# B&R Automation Studio project Panasonic_LinkaKapacitorov_A2021040 (part 3)

#### OvlRucnejCitackyQR.st
```iecst
ACTION OvlRucnejCitackyQR:

	//"$L"  LF - linefeed - skok na druhý riadok

	CASE RucCitackaQR.Step OF

		0://Nulovanie//
			RucCitackaQR.Command.PrimajData:= FALSE;
			RucCitackaQR.Command.ZatvorKomunikaciu:= FALSE;
			RucCitackaQR.Command.PotvrdeniePoruchy:= FALSE;
			RucCitackaQR.Status.PoruchaOtvoreniaKomunikacie:= FALSE;
			RucCitackaQR.Status.PoruchaZatvoreniaKomunikacie:= FALSE;
			RucCitackaQR.Status.PoruchaCitaniaDat:= FALSE;
			RucCitackaQR.Status.PoruchaUvolneniaRECEIVE_Buffera:= FALSE;
			RucCitackaQR.Step:= 1;

		1://Rozhodnutie o činnosti//
			IF RucCitackaQR.Command.PrimajData THEN
				RucCitackaQR.Step:= 10;
			ELSIF Linka.CitackaQRkodu_AKTIVNA THEN
				RucCitackaQR.Step:= 10;
			END_IF

		10://Prímanie dát - otvorenie seriovej komunikácie//
			RucCitackaQR.FRM_xopen_0.enable:= TRUE;
			RucCitackaQR.FRM_xopen_0.device:=  ADR('IF1');
			RucCitackaQR.FRM_xopen_0.mode:= ADR('/PHY=RS232 /BD=115200 /DB=8 /PA=N /SB=1');
			RucCitackaQR.FRM_xopen_0.config:= ADR(RucCitackaQR.xopenConfig);

			RucCitackaQR.xopenConfig.idle:= 100;
			RucCitackaQR.xopenConfig.delimc:= 0;
			RucCitackaQR.xopenConfig.delim[0]:= 0;
			RucCitackaQR.xopenConfig.delim[1]:= 0;
			RucCitackaQR.xopenConfig.tx_cnt:= 3;
			RucCitackaQR.xopenConfig.rx_cnt:= 3;
			RucCitackaQR.xopenConfig.tx_len:= 256;
			RucCitackaQR.xopenConfig.rx_len:= 256;
			RucCitackaQR.xopenConfig.argc:= 0;
			RucCitackaQR.xopenConfig.argv:= 0;

			RucCitackaQR.FRM_xopen_0();

			IF RucCitackaQR.FRM_xopen_0.status = 0 THEN   //Otvorenie komunikácie prebehlo OK
				RucCitackaQR.Step:= 11;
			ELSIF RucCitackaQR.FRM_xopen_0.status = 65535 THEN  //Prebieha otvorenie komunikácie - stav BUSY
				RucCitackaQR.Step:= 10;
			ELSE
				RucCitackaQR.Status.PoruchaOtvoreniaKomunikacie:= TRUE;
				RucCitackaQR.Step:= 100;  //Porucha otvorenia komunikácie
			END_IF

		11://Prímanie dát - čítanie dát z komunikácie//
			RucCitackaQR.FRM_read_0.enable:= TRUE;
			RucCitackaQR.FRM_read_0.ident:= RucCitackaQR.FRM_xopen_0.ident;
			RucCitackaQR.FRM_read_0();

			IF RucCitackaQR.FRM_read_0.status = 0 THEN //Čítanie dát z komunikácie prebehlo OK
				RucCitackaQR.Step:= 12;
			ELSIF RucCitackaQR.Command.ZatvorKomunikaciu THEN
				RucCitackaQR.Step:= 0;
			ELSIF NOT Linka.CitackaQRkodu_AKTIVNA THEN
				RucCitackaQR.Step:= 0;
			ELSIF RucCitackaQR.FRM_read_0.status = 60 THEN //Prebieha čítanie dát z komunikácie - stav žiadne dáta
				RucCitackaQR.Step:= 11;
			ELSIF RucCitackaQR.FRM_read_0.status = 8079 THEN //Prišli zlé alebo neúplné dáta
				RucCitackaQR.Step:= 18;
			ELSE
				RucCitackaQR.Status.PoruchaCitaniaDat:= TRUE;
				RucCitackaQR.Step:= 100;  //Porucha čítania dát z komunikácie
			END_IF

		12://Prímanie dát - kopírovanie dát do RECEIVE buffera//
			brsmemset(ADR(RucCitackaQR.PrecitaneData),0,SIZEOF(RucCitackaQR.PrecitaneData)); //Vynulovanie prečítanej správy
			brsmemcpy(ADR(RucCitackaQR.PrecitaneData),RucCitackaQR.FRM_read_0.buffer,RucCitackaQR.FRM_read_0.buflng); //Zkopírovanie dát z RECEIVE buffera do prečítanej správy
			RucCitackaQR.Step:= 18;

		18://Prímanie dát - uvolnenie RECEIVE buffera//
			RucCitackaQR.FRM_rbuf_0.enable:= TRUE;
			RucCitackaQR.FRM_rbuf_0.buffer:= RucCitackaQR.FRM_read_0.buffer;
			RucCitackaQR.FRM_rbuf_0.buflng:= RucCitackaQR.FRM_read_0.buflng;
			RucCitackaQR.FRM_rbuf_0.ident:= RucCitackaQR.FRM_xopen_0.ident;
			RucCitackaQR.FRM_rbuf_0();

			IF RucCitackaQR.FRM_rbuf_0.status = 0 THEN //Uvolnenie RECEIVE buffera prebehlo OK
				IF RucCitackaQR.Command.ZatvorKomunikaciu THEN
					RucCitackaQR.Step:= 20;
				ELSE
					RucCitackaQR.Step:= 11;
				END_IF
			ELSIF RucCitackaQR.FRM_rbuf_0.status = 65535 THEN //Prebieha uvolnenie RECEIVE buffera - stav BUSY
				RucCitackaQR.Step:= 18;
			ELSIF RucCitackaQR.FRM_rbuf_0.status = 8072 THEN //Buffer je poškodený - op)tovné čítanie
				RucCitackaQR.Step:= 11;
			ELSE
				RucCitackaQR.Status.PoruchaUvolneniaRECEIVE_Buffera:= TRUE;
				RucCitackaQR.Step:= 100;  //Porucha uvolnenia RECEIVE buffera
			END_IF

		20://Prímanie dát - zatvorenie komunikácie//
			RucCitackaQR.FRM_close_0.enable:= TRUE;
			RucCitackaQR.FRM_close_0.ident:= RucCitackaQR.FRM_xopen_0.ident;
			RucCitackaQR.FRM_close_0();

			IF RucCitackaQR.FRM_close_0.status = 0 THEN //Zatvorenie komunikácie prebehlo OK
				RucCitackaQR.Step:= 0;
			ELSIF RucCitackaQR.FRM_close_0.status = 65535 THEN //Prebieha zatvorenie komunikácie - stav BUSY
				RucCitackaQR.Step:= 20;
			ELSE
				RucCitackaQR.Status.PoruchaZatvoreniaKomunikacie:= TRUE;
				RucCitackaQR.Step:= 100;  //Porucha zatvorenia komunikácie
			END_IF

		100://Porucha komunikácie//
			IF RucCitackaQR.Command.PotvrdeniePoruchy THEN
				RucCitackaQR.Step:= 0;
			END_IF

	END_CASE

END_ACTION
```

#### ZmenaModelu.st
```iecst
ACTION ZmenaModelu:

		//***********************************************Zobrazenie stavov zmeny modelu***********************************************//
    //0 - Čakám na zmenu modelu.
    //1 - Nebol načítaný názov modelu !!!
    //2 - Nebol načítaný LOT !!!
    //3 - Zmena modelu prebehla OK !!!
	//4 - Zadaný model nieje v databázi linky !!!

	//Farba pozadia//
	//0 - sivá
	//1 - modrá
	//2 - zelená
	//3 - červená

	IF EDGEPOS(Vizu.CisloAktualnejObrazovky = 4)THEN
		Vizu.StavZmenyModelu_Index:= 0;
		Vizu.StavZmenyModelu_Farba:= 0;
		Vizu.Nacitany_MODEL:= '';
		Vizu.Nacitany_LOT:= '';
	END_IF

	//Zistenie počtu načítaných znakov//
	PocetNacitanychZnakov := brsstrlen(ADR(RucCitackaQR.PrecitaneData)); //Zistenie počtu znakov vstupnej spravy

	//Zistenie či sa jedná o Názov modelu alebo číslo Lotu//
	brsmemcpy(ADR(NacitaneZnaky_POLE),ADR(RucCitackaQR.PrecitaneData),SIZEOF(RucCitackaQR.PrecitaneData)); //Vyplnenie polia znakmy vstupnej správy

	//Zapísanie načítanej hodnoty do pola Nazov Modelu alebo Cislo Lotu// EZT
	IF RucCitackaQR.PrecitaneData <> '' THEN
		IF NacitaneZnaky_POLE[0] = 69 AND NacitaneZnaky_POLE[1] = 90 AND NacitaneZnaky_POLE[2] = 84 AND PocetNacitanychZnakov = 12 THEN
			Vizu.Nacitany_MODEL:= RucCitackaQR.PrecitaneData;
		ELSIF NacitaneZnaky_POLE[0] = 66 AND PocetNacitanychZnakov = 11 THEN
			Vizu.Nacitany_LOT:= RucCitackaQR.PrecitaneData;
		END_IF
		RucCitackaQR.PrecitaneData:= '';
	END_IF

	CASE SC_ZmenaModelu.Step OF

		0://Vynulovanie uživatela//
			SC_ZmenaModelu.StepName:= '0 - Nulovanie';
			Linka.ZmenModel:= FALSE;
			i:= 0;
			SC_ZmenaModelu.ResetStep:= TRUE;
			SC_ZmenaModelu.Step:= 1;

		1://Rozhodnutie o činnosti//
			SC_ZmenaModelu.StepName:= '1 - Rozhodnutie o cinnosti';
			IF Linka.ZmenModel THEN
				SC_ZmenaModelu.Step:= 10;
			END_IF

		10://Kontrola zadania modelu//
			SC_ZmenaModelu.StepName:= '10 - Kontrola zadania modelu';
			IF Vizu.Nacitany_MODEL <> '' AND Vizu.Nacitany_LOT <> '' THEN
				SC_ZmenaModelu.ResetStep:= TRUE;
				SC_ZmenaModelu.Step:= 11;
			ELSE
				IF Vizu.Nacitany_MODEL = '' THEN
					Vizu.StavZmenyModelu_Index:= 1;
					Vizu.StavZmenyModelu_Farba:= 3;
				ELSIF Vizu.Nacitany_LOT = '' THEN
					Vizu.StavZmenyModelu_Index:= 2;
					Vizu.StavZmenyModelu_Farba:= 3;
				END_IF
				SC_ZmenaModelu.ResetStep:= TRUE;
				SC_ZmenaModelu.Step:= 0;
			END_IF

		11://Hladanie modelu v recepturach//
			SC_ZmenaModelu.StepName:= '11 - Hladanie modelu v recepturach';
			ModelNajdeny:= FALSE;
			FOR i:= 0 TO 150 BY 1 DO
				IF (Receptura[i].NazovModelu = Vizu.Nacitany_MODEL) AND NOT ModelNajdeny THEN
					HistoriaVyroby[IndexHistorie].NazovModelu:= Zvoleny_MODEL;
					HistoriaVyroby[IndexHistorie].NazovLOTU:= Zvoleny_LOT;
					HistoriaVyroby[IndexHistorie].PocetVyrobenychKusov_OK:= PocetVyrobenychKusov_OK;
					HistoriaVyroby[IndexHistorie].PocetVyrobenychKusov_NG:= PocetVyrobenychKusov_NG;
					HistoriaVyroby[IndexHistorie].Pomer_OK_kusov_IDR:= Pomer_OK_kusov_IDR;
					IndexHistorie:= IndexHistorie + 1;
					IF IndexHistorie > 5 THEN
						IndexHistorie:= 0;
					END_IF
					Linka.PAR.Zvoleny_MODEL:= Vizu.Nacitany_MODEL;
					Zvoleny_MODEL:= Vizu.Nacitany_MODEL;
					Linka.PAR.Zvoleny_LOT:= Vizu.Nacitany_LOT;
					Zvoleny_LOT:= Vizu.Nacitany_LOT;
					Linka.PAR.IndexZvoleneReceptury:= i;
					Vizu.StavZmenyModelu_Index:= 3;
					Vizu.StavZmenyModelu_Farba:= 2;
					RESET_PoctuVyrobenychKusov:= TRUE;
					Linka.Rezim_BezCistenia:= FALSE;
					Linka.Rezim_BezTlaceEtikety:= FALSE;
					Linka.Rezim_Testovania:= FALSE;
					NacitajRecepturu:= TRUE;
					ModelNajdeny:= TRUE;
				END_IF
			END_FOR
			IF NOT ModelNajdeny THEN
				Vizu.StavZmenyModelu_Index:= 4;
				Vizu.StavZmenyModelu_Farba:= 3;
			END_IF
			SC_ZmenaModelu.ResetStep:= TRUE;
			SC_ZmenaModelu.Step:= 0;

	END_CASE

END_ACTION
```

### Program Logical/Program/KontrolaOtacaniaTrysiek (IEC)

#### Main.st - Init, cyclic, exit code
```iecst
PROGRAM _INIT
	(* Insert code here *)

END_PROGRAM

PROGRAM _CYCLIC

	//Volanie funkcie SequenceControl//
	SequenceControl(SC:= SC_OvlCistenia);

	CASE SC_OvlCistenia.Step OF

		0:
			SC_OvlCistenia.StepName:='0 - Nulovanie';
			CasOtacaniaHornejTrisky_1.IN:= FALSE;
			CasOtacaniaHornejTrisky_2.IN:= FALSE;
			CasOtacaniaHornejTrisky_3.IN:= FALSE;
			CasOtacaniaHornejTrisky_4.IN:= FALSE;
			CasOtacaniaSpodnejTrisky_1.IN:= FALSE;
			CasOtacaniaSpodnejTrisky_2.IN:= FALSE;
			CasOtacaniaSpodnejTrisky_3.IN:= FALSE;
			Linka.OUT.IonJednotka_START:= FALSE;
			Linka.OUT.IonJednotka_AIR:= FALSE;
			SC_OvlCistenia.ResetStep:= TRUE;
			SC_OvlCistenia.Step:= 1;

		1:
			SC_OvlCistenia.StepName:='1 - Cakam na spustenie cistenia';

			IF Linka.OUT.IonJednotka_START THEN
				SC_OvlCistenia.Step:= 10;
			END_IF

		10:
			SC_OvlCistenia.StepName:='10 - spustenie kontroly otacania trisiek';
			SC_OvlCistenia.IdleTime.PT:= T#2s;
			SC_OvlCistenia.AlarmTime.PT:= T#1s;

			Linka.OUT.IonJednotka_AIR:= TRUE;

			SC_OvlCistenia.IdleTime.IN:= TRUE;

			IF EDGE(Linka.IN.SnimacRotacieHornTrysiek_1_IS7) THEN
				CasOtacaniaHornejTrisky_1.IN:= FALSE;
			ELSE
				CasOtacaniaHornejTrisky_1.IN:= TRUE;
			END_IF

			IF EDGE(Linka.IN.SnimacRotacieHornTrysiek_2_IS8) THEN
				CasOtacaniaHornejTrisky_2.IN:= FALSE;
			ELSE
				CasOtacaniaHornejTrisky_2.IN:= TRUE;
			END_IF

			IF EDGE(Linka.IN.SnimacRotacieHornTrysiek_3_IS9) THEN
				CasOtacaniaHornejTrisky_3.IN:= FALSE;
			ELSE
				CasOtacaniaHornejTrisky_3.IN:= TRUE;
			END_IF

			IF EDGE(Linka.IN.SnimacRotacieHornTrysiek_4_IS10) THEN
				CasOtacaniaHornejTrisky_4.IN:= FALSE;
			ELSE
				CasOtacaniaHornejTrisky_4.IN:= TRUE;
			END_IF

			IF EDGE(Linka.IN.SnimacRotacieSpodTrysiek_1_IS11) THEN
				CasOtacaniaSpodnejTrisky_1.IN:= FALSE;
			ELSE
				CasOtacaniaSpodnejTrisky_1.IN:= TRUE;
			END_IF

			IF EDGE(Linka.IN.SnimacRotacieSpodTrysiek_2_IS12) THEN
				CasOtacaniaSpodnejTrisky_2.IN:= FALSE;
			ELSE
				CasOtacaniaSpodnejTrisky_2.IN:= TRUE;
			END_IF

			IF EDGE(Linka.IN.SnimacRotacieSpodTrysiek_3_IS13) THEN
				CasOtacaniaSpodnejTrisky_3.IN:= FALSE;
			ELSE
				CasOtacaniaSpodnejTrisky_3.IN:= TRUE;
			END_IF

			IF NOT Linka.OUT.IonJednotka_START THEN
				SC_OvlCistenia.ResetStep:= TRUE;
				SC_OvlCistenia.Step:= 0;
			END_IF

			IF SC_OvlCistenia.IdleTime.Q THEN
				IF CasOtacaniaHornejTrisky_1.Q THEN
					Alarmy[37]:= TRUE;
					Linka.STAV.PoruchaOtacaniaTrysiek:= TRUE;
					SC_OvlCistenia.ResetStep:= TRUE;
					SC_OvlCistenia.Step:= 0;
				ELSIF CasOtacaniaHornejTrisky_2.Q THEN
					Alarmy[37]:= TRUE;
					Linka.STAV.PoruchaOtacaniaTrysiek:= TRUE;
					SC_OvlCistenia.ResetStep:= TRUE;
					SC_OvlCistenia.Step:= 0;
				ELSIF CasOtacaniaHornejTrisky_3.Q THEN
					Alarmy[37]:= TRUE;
					Linka.STAV.PoruchaOtacaniaTrysiek:= TRUE;
					SC_OvlCistenia.ResetStep:= TRUE;
					SC_OvlCistenia.Step:= 0;
				ELSIF CasOtacaniaHornejTrisky_4.Q THEN
					Alarmy[37]:= TRUE;
					Linka.STAV.PoruchaOtacaniaTrysiek:= TRUE;
					SC_OvlCistenia.ResetStep:= TRUE;
					SC_OvlCistenia.Step:= 0;
				ELSIF CasOtacaniaSpodnejTrisky_1.Q THEN
					Alarmy[38]:= TRUE;
					Linka.STAV.PoruchaOtacaniaTrysiek:= TRUE;
					SC_OvlCistenia.ResetStep:= TRUE;
					SC_OvlCistenia.Step:= 0;
				ELSIF CasOtacaniaSpodnejTrisky_2.Q THEN
					Alarmy[38]:= TRUE;
					Linka.STAV.PoruchaOtacaniaTrysiek:= TRUE;
					SC_OvlCistenia.ResetStep:= TRUE;
					SC_OvlCistenia.Step:= 0;
				ELSIF CasOtacaniaSpodnejTrisky_3.Q THEN
					Alarmy[38]:= TRUE;
					Linka.STAV.PoruchaOtacaniaTrysiek:= TRUE;
					SC_OvlCistenia.ResetStep:= TRUE;
					SC_OvlCistenia.Step:= 0;
				END_IF
			END_IF

	END_CASE

	CasOtacaniaHornejTrisky_1.PT:= T#300ms;
	CasOtacaniaHornejTrisky_1();
	CasOtacaniaHornejTrisky_2.PT:= T#300ms;
	CasOtacaniaHornejTrisky_2();
	CasOtacaniaHornejTrisky_3.PT:= T#300ms;
	CasOtacaniaHornejTrisky_3();
	CasOtacaniaHornejTrisky_4.PT:= T#300ms;
	CasOtacaniaHornejTrisky_4();
	CasOtacaniaSpodnejTrisky_1.PT:= T#500ms;
	CasOtacaniaSpodnejTrisky_1();
	CasOtacaniaSpodnejTrisky_2.PT:= T#500ms;
	CasOtacaniaSpodnejTrisky_2();
	CasOtacaniaSpodnejTrisky_3.PT:= T#500ms;
	CasOtacaniaSpodnejTrisky_3();

END_PROGRAM

PROGRAM _EXIT
	(* Insert code here *)

END_PROGRAM
```

#### Variables.var - Local variables
```iecst
VAR
	SC_OvlCistenia : SequenceControlTyp := (0);
	CasOtacaniaHornejTrisky_1 : TON := (0);
	CasOtacaniaHornejTrisky_2 : TON := (0);
	CasOtacaniaHornejTrisky_3 : TON := (0);
	CasOtacaniaHornejTrisky_4 : TON := (0);
	CasOtacaniaSpodnejTrisky_1 : TON := (0);
	CasOtacaniaSpodnejTrisky_2 : TON := (0);
	CasOtacaniaSpodnejTrisky_3 : TON := (0);
END_VAR
```

### Program Logical/Program/VstupnyVytah (IEC)

#### Main.st - Init, cyclic, exit code
```iecst
PROGRAM _INIT
	VstupVytah.PAR.Zdvih_ZadanaJoggRychlost:= 10;

END_PROGRAM

PROGRAM _CYCLIC

	//Volanie podprogramov//
	OvlMenica;
	OvlDveri;
	OvlCitackyRFID;

	//Volanie funkcie SequenceControl//
	SequenceControl(SC:= SC_VstupVytah);

	//Reset sekcie //
	IF VstupVytah.Reset THEN
		SC_VstupVytah.Step:= 0;
		VstupVytah.Reset:= FALSE;
	ELSIF NOT Safety.STAV.ZonaCS_AKTIVNA THEN
		SC_VstupVytah.Step:= 0;
	END_IF

	CASE SC_VstupVytah.Step OF

		0:
			SC_VstupVytah.StepName:='0 - Nulovanie';
			VstupVytah.Automat:= FALSE;
			VstupVytah.KoniecCyklu:= FALSE;
			VstupVytah.Manual:= FALSE;
			VstupVytah.STAV.PoINIT:= FALSE;
			SC_OvlMenica.Step:= 0;
			SC_OvlDveri.Step:= 0;
			VstupVytah.OUT.Dopravnik_ChodVPRED_ELR1:= FALSE;
			VstupVytah.OUT.Dopravnik_ChodVZAD_ELR1:= FALSE;
			VstupVytah.RR_Dopravnik_VPRED:= FALSE;
			VstupVytah.RR_Dopravnik_VZAD:= FALSE;
			IF PoruchaVstupnehoVytahu THEN
				VstupVytah.OUT.Banner_CervenaLED_IOS1:= Blikac200ms;
			ELSE
				VstupVytah.OUT.Banner_CervenaLED_IOS1:= FALSE;
			END_IF
			VstupVytah.OUT.Banner_ZelenaLED_IOS1:= FALSE;
			VstupVytah.STAV.PrebiehaVyvazaniePaletky:= FALSE;
			VstupVytah.STAV.VytahNapolohovany:= FALSE;
			Vizu.ZobrazHlasenie_NespravTypPaletky:= 1;
			VstupVytah.STAV.ObsluhaPotvrdilaBanner:= FALSE;
			VstupnyVytah_Statistika.IN.START_MeraniaCasu:= FALSE;

			IF Safety.STAV.ZonaCS_AKTIVNA AND Safety.STAV.ZonaVstupnyVytah_AKTIVNA AND Linka.IN.TlakVzduchu_OK_S2 AND NOT NastalaPorucha AND Linka.STAV.Hardware_OK THEN
				VstupVytah.OUT.Banner_CervenaLED_IOS1:= FALSE;
				SC_VstupVytah.ResetStep:= TRUE;
				SC_VstupVytah.Step:= 1;
			END_IF

		1:
			SC_VstupVytah.StepName:='1 - Cakam na spustenie vyroby';
			VstupVytah.KoniecCyklu:= FALSE;
			IF VstupVytah.Automat THEN
				SC_VstupVytah.Step:= 2;
			ELSIF VstupVytah.Manual THEN
				SC_VstupVytah.Step:= 700;
			END_IF

			//********************************************************Inicializácia****************************************************************************//

		2:
			SC_VstupVytah.StepName:='2 - Inicializacia - cakam na spustenie inicializacie';
			SC_VstupVytah.IdleTime.PT:= T#500ms;
			SC_VstupVytah.AlarmTime.PT:= T#5s;

			SC_VstupVytah.IdleTime.IN:= TRUE;

			IF SC_VstupVytah.IdleTime.Q THEN
				SC_VstupVytah.ResetStep:= TRUE;
				SC_VstupVytah.Step:= 5;
			END_IF

		5:
			SC_VstupVytah.StepName:='5 - Inicializacia - spustam dopravnik vytahu pre navezenie paletky';
			SC_VstupVytah.IdleTime.PT:= T#500ms;
			SC_VstupVytah.AlarmTime.PT:= T#7s;

			SC_VstupVytah.IdleTime.IN:= VstupVytah.IN.PritomnostPaletky_IS3;

			IF NOT SC_VstupVytah.Switch1 THEN
				VstupVytah.OUT.Dopravnik_ChodVZAD_ELR1:= TRUE;
				SC_VstupVytah.AlarmTime.IN:= TRUE;
				SC_VstupVytah.Switch1:= TRUE;
			END_IF

			IF SC_VstupVytah.IdleTime.Q AND NOT VstupVytah.IN.PrechodDopravnikaVytahu_OS1 THEN
				VstupVytah.OUT.Dopravnik_ChodVZAD_ELR1:= FALSE;
				SC_VstupVytah.ResetStep:= TRUE;
				SC_VstupVytah.Step:= 10;
			ELSIF SC_VstupVytah.AlarmTime.Q AND NOT VstupVytah.IN.PritomnostPaletky_IS3 AND NOT VstupVytah.IN.PrechodDopravnikaVytahu_OS1 THEN
				VstupVytah.OUT.Dopravnik_ChodVZAD_ELR1:= FALSE;
				SC_VstupVytah.ResetStep:= TRUE;
				SC_VstupVytah.Step:= 10;
			ELSIF SC_VstupVytah.AlarmTime.Q AND VstupVytah.IN.PrechodDopravnikaVytahu_OS1 THEN
				Alarmy[44]:= TRUE;
				PoruchaVstupnehoVytahu:= TRUE;
				SC_VstupVytah.ResetStep:= TRUE;
				SC_VstupVytah.Step:= 0;
			END_IF

		10:
			SC_VstupVytah.StepName:='10 - Inicializacia - kontrola zatvorenia dveri vytahu';
			SC_VstupVytah.IdleTime.PT:= T#500ms;
			SC_VstupVytah.AlarmTime.PT:= T#7s;

			IF VstupVytah.IN.DvereVytahuZatvorene_MS2 THEN
				SC_VstupVytah.ResetStep:= TRUE;
				SC_VstupVytah.Step:= 15;
			ELSE
				SC_VstupVytah.ResetStep:= TRUE;
				SC_VstupVytah.Step:= 13;
			END_IF

		13:
			SC_VstupVytah.StepName:='10 - Inicializacia - zatvorenie dveri vytahu';
			SC_VstupVytah.IdleTime.PT:= T#500ms;
			SC_VstupVytah.AlarmTime.PT:= T#7s;

			IF NOT SC_VstupVytah.Switch1 THEN
				Dvere_ZATVOR:= TRUE;
				SC_VstupVytah.Switch1:= TRUE;
			END_IF

			IF VstupVytah.IN.DvereVytahuZatvorene_MS2 THEN
				SC_VstupVytah.ResetStep:= TRUE;
				SC_VstupVytah.Step:= 15;
			END_IF

		15:
			SC_VstupVytah.StepName:='15 - Inicializacia - kontrola homingu zdvihu vytahu';
			SC_VstupVytah.IdleTime.PT:= T#2s;
			SC_VstupVytah.AlarmTime.PT:= T#5s;

			IF VstupVytah.STAV.Zdvih_HomingOK THEN
				SC_VstupVytah.ResetStep:= TRUE;
				SC_VstupVytah.Step:= 35;
			ELSE
				SC_VstupVytah.ResetStep:= TRUE;
				SC_VstupVytah.Step:= 18;
			END_IF

		18:
			SC_VstupVytah.StepName:='18 - Inicializacia - cakam na spustenie homingu zdvihu vytahu';
			SC_VstupVytah.IdleTime.PT:= T#1s;
			SC_VstupVytah.AlarmTime.PT:= T#5s;

			SC_VstupVytah.IdleTime.IN:= Safety.STAV.BarieraVstupVytahu_AKTIVNA AND NOT VstupVytah.IN.PrechodDopravnikaVytahu_OS1;

			IF SC_VstupVytah.IdleTime.Q THEN
				SC_VstupVytah.ResetStep:= TRUE;
				SC_VstupVytah.Step:= 20;
			END_IF

		20:
			SC_VstupVytah.StepName:='20 - Inicializacia - spustam homing zdvihu vytahu';
			SC_VstupVytah.IdleTime.PT:= T#2s;
			SC_VstupVytah.AlarmTime.PT:= T#5s;

			VstupVytah.OUT.Banner_CervenaLED_IOS1:= TRUE;

			IF NOT SC_VstupVytah.Switch1 THEN
				Zdvih_HOME:= TRUE;
				SC_VstupVytah.Switch1:= TRUE;
			END_IF

			IF VstupVytah.STAV.Zdvih_HomingOK THEN
				SC_VstupVytah.ResetStep:= TRUE;
				SC_VstupVytah.Step:= 35;
			ELSIF NOT Safety.STAV.BarieraVstupVytahu_AKTIVNA THEN
				Alarmy[46]:= TRUE;
				PoruchaVstupnehoVytahu:= TRUE;
				SC_VstupVytah.ResetStep:= TRUE;
				SC_VstupVytah.Step:= 0;
			ELSIF VstupVytah.IN.PrechodDopravnikaVytahu_OS1 THEN
				Alarmy[47]:= TRUE;
				PoruchaVstupnehoVytahu:= TRUE;
				SC_VstupVytah.ResetStep:= TRUE;
				SC_VstupVytah.Step:= 0;
			END_IF

		35:
			SC_VstupVytah.StepName:='35 - Inicializacia - cakam na spustenie presunu vytahu do hornej pozicie vyvazania';
			SC_VstupVytah.IdleTime.PT:= T#1s;
			SC_VstupVytah.AlarmTime.PT:= T#5s;

			SC_VstupVytah.IdleTime.IN:= Safety.STAV.BarieraVstupVytahu_AKTIVNA AND NOT VstupVytah.IN.PrechodDopravnikaVytahu_OS1;

			IF SC_VstupVytah.IdleTime.Q THEN
				SC_VstupVytah.ResetStep:= TRUE;
				SC_VstupVytah.Step:= 38;
			END_IF

		38:
			SC_VstupVytah.StepName:='38 - Inicializacia - presuvam vytah do hornej pozicie vyvazania';
			SC_VstupVytah.IdleTime.PT:= T#1s;
			SC_VstupVytah.AlarmTime.PT:= T#5s;

			VstupVytah.OUT.Banner_CervenaLED_IOS1:= TRUE;
			VstupVytah.PAR.Zdvih_ZadanaRychlost:= 50;
			VstupVytah.PAR.Zdvih_ZadanaPozicia:= RemPremenne.VstupVytah_PozVyvazania;

			IF NOT SC_VstupVytah.Switch1 AND SC_OvlMenica.Step = 1 THEN
				Zdvih_POLOHUJ:= TRUE;
				SC_VstupVytah.Switch1:= TRUE;
			END_IF

			IF VstupVytah.STAV.VytahNapolohovany THEN
				VstupVytah.STAV.VytahNapolohovany:= FALSE;
				VstupVytah.OUT.Banner_CervenaLED_IOS1:= FALSE;
				SC_VstupVytah.ResetStep:= TRUE;
				SC_VstupVytah.Step:= 40;
			ELSIF NOT Safety.STAV.BarieraVstupVytahu_AKTIVNA THEN
				Alarmy[46]:= TRUE;
				PoruchaVstupnehoVytahu:= TRUE;
				SC_VstupVytah.ResetStep:= TRUE;
				SC_VstupVytah.Step:= 0;
			ELSIF VstupVytah.IN.PrechodDopravnikaVytahu_OS1 THEN
				Alarmy[47]:= TRUE;
				PoruchaVstupnehoVytahu:= TRUE;
				SC_VstupVytah.ResetStep:= TRUE;
				SC_VstupVytah.Step:= 0;
			END_IF

		40:
			SC_VstupVytah.StepName:='40 - Inicializacia - kontrola pritomnosti paletky na dopravniku vytahu';
			SC_VstupVytah.IdleTime.PT:= T#2s;
			SC_VstupVytah.AlarmTime.PT:= T#5s;

			IF VstupVytah.IN.PritomnostPaletky_IS3 THEN
				VstupVytah.STAV.PoINIT := TRUE;
				SC_VstupVytah.ResetStep:= TRUE;
				SC_VstupVytah.Step:= 100;
			ELSE
				VstupVytah.STAV.PoINIT := TRUE;
				SC_VstupVytah.ResetStep:= TRUE;
				SC_VstupVytah.Step:= 100;
			END_IF

			//********************************************************Automatický režim****************************************************************************//

		100:
			SC_VstupVytah.StepName:='100 - Automaticky Rezim - cakam na navezenie paletky na vytah zo spodneho vratneho dopravnika';
			SC_VstupVytah.IdleTime.PT:= T#500ms;
			SC_VstupVytah.AlarmTime.PT:= T#5s;

			IF VstupVytah.KoniecCyklu THEN
				SC_VstupVytah.ResetStep:= TRUE;
				SC_VstupVytah.Step:= 0;
			ELSIF SC_StoperVratDopravnika.Step = 101 AND NOT VstupVytah.IN.PritomnostPaletky_IS3 AND NOT VstupVytah.IN.PrechodDopravnikaVytahu_OS1 AND Safety.STAV.BarieraVstupVytahu_AKTIVNA AND VstupVytah.IN.DvereVytahuZatvorene_MS2 THEN
				SC_VstupVytah.ResetStep:= TRUE;
				SC_VstupVytah.Step:= 103;
			ELSIF VstupVytah.IN.PritomnostPaletky_IS3 AND Safety.STAV.BarieraVstupVytahu_AKTIVNA THEN
				SC_VstupVytah.ResetStep:= TRUE;
				SC_VstupVytah.Step:= 111;
			END_IF

		103:
			SC_VstupVytah.StepName:='103 - Automaticky Rezim - presuvam vytah do spodnej pozicie navazania';
			SC_VstupVytah.IdleTime.PT:= T#1s;
			SC_VstupVytah.AlarmTime.PT:= T#5s;

			VstupVytah.OUT.Banner_CervenaLED_IOS1:= TRUE;
			VstupVytah.PAR.Zdvih_ZadanaRychlost:= 50;
			VstupVytah.PAR.Zdvih_ZadanaPozicia:= RemPremenne.VstupVytah_PozNavazania;

			IF NOT SC_VstupVytah.Switch1 AND SC_OvlMenica.Step = 1 THEN
				Zdvih_POLOHUJ:= TRUE;
				VstupVytah.OUT.Dopravnik_ChodVZAD_ELR1:= TRUE;
				SC_VstupVytah.Switch1:= TRUE;
			END_IF

			IF VstupVytah.STAV.VytahNapolohovany THEN
				VstupVytah.STAV.VytahNapolohovany:= FALSE;
				VstupVytah.OUT.Dopravnik_ChodVZAD_ELR1:= FALSE;
				SC_VstupVytah.ResetStep:= TRUE;
				SC_VstupVytah.Step:= 105;
			ELSIF NOT Safety.STAV.BarieraVstupVytahu_AKTIVNA THEN
				Alarmy[46]:= TRUE;
				PoruchaVstupnehoVytahu:= TRUE;
				SC_VstupVytah.ResetStep:= TRUE;
				SC_VstupVytah.Step:= 0;
			ELSIF VstupVytah.IN.PrechodDopravnikaVytahu_OS1 THEN
				Alarmy[47]:= TRUE;
				PoruchaVstupnehoVytahu:= TRUE;
				SC_VstupVytah.ResetStep:= TRUE;
				SC_VstupVytah.Step:= 0;
			END_IF

		105:
			SC_VstupVytah.StepName:='105 - Automaticky Rezim - navazam paletku na dopravnik vytahu';
			SC_VstupVytah.IdleTime.PT:= T#200ms;
			SC_VstupVytah.AlarmTime.PT:= T#20s;

			SC_VstupVytah.IdleTime.IN:= VstupVytah.IN.PritomnostPaletky_IS3;

			IF NOT SC_VstupVytah.Switch1 THEN
				VstupVytah.OUT.Dopravnik_ChodVZAD_ELR1:= TRUE;
				SC_VstupVytah.AlarmTime.IN:= TRUE;
				SC_VstupVytah.Switch1:= TRUE;
			END_IF

			IF SC_VstupVytah.IdleTime.Q AND NOT VstupVytah.IN.PrechodDopravnikaVytahu_OS1 THEN
				VstupVytah.OUT.Dopravnik_ChodVZAD_ELR1:= FALSE;
				SC_VstupVytah.ResetStep:= TRUE;
				SC_VstupVytah.Step:= 108;
			ELSIF SC_VstupVytah.AlarmTime.Q THEN
				Alarmy[45]:= TRUE;
				PoruchaVstupnehoVytahu:= TRUE;
				SC_VstupVytah.ResetStep:= TRUE;
				SC_VstupVytah.Step:= 0;
			END_IF

		108:
			SC_VstupVytah.StepName:='108 - Automaticky Rezim - cakam na presun vytahu do hornej pozicie vyvazania';
			SC_VstupVytah.IdleTime.PT:= T#500ms;
			SC_VstupVytah.AlarmTime.PT:= T#10s;

			SC_VstupVytah.IdleTime.IN:= Safety.STAV.BarieraVstupVytahu_AKTIVNA AND NOT VstupVytah.IN.PrechodDopravnikaVytahu_OS1 AND VstupVytah.IN.DvereVytahuZatvorene_MS2;

			IF SC_VstupVytah.IdleTime.Q THEN
				SC_VstupVytah.ResetStep:= TRUE;
				SC_VstupVytah.Step:= 110;
			END_IF

		110:
			SC_VstupVytah.StepName:='110 - Automaticky Rezim - presuvam vytah do hornej pozicie vyvazania';
			SC_VstupVytah.IdleTime.PT:= T#500ms;
			SC_VstupVytah.AlarmTime.PT:= T#10s;

			VstupVytah.OUT.Banner_CervenaLED_IOS1:= TRUE;
			VstupVytah.PAR.Zdvih_ZadanaRychlost:= 50;
			VstupVytah.PAR.Zdvih_ZadanaPozicia:= RemPremenne.VstupVytah_PozVyvazania;

			IF NOT SC_VstupVytah.Switch1 AND SC_OvlMenica.Step = 1 THEN
				Zdvih_POLOHUJ:= TRUE;
				SC_VstupVytah.Switch1:= TRUE;
			END_IF

			IF VstupVytah.STAV.VytahNapolohovany THEN
				VstupVytah.STAV.VytahNapolohovany:= FALSE;
				SC_VstupVytah.ResetStep:= TRUE;
				SC_VstupVytah.Step:= 111;
			ELSIF NOT Safety.STAV.BarieraVstupVytahu_AKTIVNA THEN
				Alarmy[46]:= TRUE;
				PoruchaVstupnehoVytahu:= TRUE;
				SC_VstupVytah.ResetStep:= TRUE;
				SC_VstupVytah.Step:= 0;
			ELSIF VstupVytah.IN.PrechodDopravnikaVytahu_OS1 THEN
				Alarmy[47]:= TRUE;
				PoruchaVstupnehoVytahu:= TRUE;
				SC_VstupVytah.ResetStep:= TRUE;
				SC_VstupVytah.Step:= 0;
			END_IF

		111:
			SC_VstupVytah.StepName:='111 - Automaticky Rezim - kontrola pritomnosti paletky';
			SC_VstupVytah.IdleTime.PT:= T#200ms;
			SC_VstupVytah.AlarmTime.PT:= T#10s;

			IF VstupVytah.IN.PritomnostPaletky_IS3 THEN
				SC_VstupVytah.ResetStep:= TRUE;
				SC_VstupVytah.Step:= 113;
			ELSE
				SC_VstupVytah.ResetStep:= TRUE;
				SC_VstupVytah.Step:= 112;
			END_IF

		112:
			SC_VstupVytah.StepName:='112 - Automaticky Rezim - hladanie paletky na dopravniku vytahu';
			SC_VstupVytah.IdleTime.PT:= T#5s;
			SC_VstupVytah.AlarmTime.PT:= T#10s;

			IF NOT SC_VstupVytah.Switch1 THEN
				VstupVytah.OUT.Dopravnik_ChodVZAD_ELR1:= TRUE;
				SC_VstupVytah.IdleTime.IN:= TRUE;
				SC_VstupVytah.Switch1:= TRUE;
			END_IF

			IF VstupVytah.IN.PritomnostPaletky_IS3 THEN
				VstupVytah.OUT.Dopravnik_ChodVZAD_ELR1:= FALSE;
				SC_VstupVytah.ResetStep:= TRUE;
				SC_VstupVytah.Step:= 111;
			ELSIF SC_VstupVytah.IdleTime.Q THEN
				VstupVytah.OUT.Dopravnik_ChodVZAD_ELR1:= FALSE;
				SC_VstupVytah.ResetStep:= TRUE;
				SC_VstupVytah.Step:= 100;
			END_IF

		113:
			SC_VstupVytah.StepName:='113 - Automaticky Rezim - citam cislo paletky a priradujem index paletky';
			SC_VstupVytah.IdleTime.PT:= T#20ms;
			SC_VstupVytah.AlarmTime.PT:= T#10s;

			SC_VstupVytah.IdleTime.IN:= RFID_Hlava_1.STAV.PritomnostCipu;

			IF SC_VstupVytah.IdleTime.Q THEN
				IF RFID_Hlava_1.PAR.PrecitaneCisloPaletky <> '' AND RFID_Hlava_1.PAR.PrecitanyTypPaletky <> '' THEN
					i:=  STRING_TO_USINT(RFID_Hlava_1.PAR.PrecitaneCisloPaletky);
					SC_VstupVytah.ResetStep:= TRUE;
					SC_VstupVytah.Step:= 115;
				ELSE
					Alarmy[60]:= TRUE;
					PoruchaVstupnehoVytahu:= TRUE;
					SC_VstupVytah.ResetStep:= TRUE;
					SC_VstupVytah.Step:= 0;
				END_IF
			END_IF

		115:
			SC_VstupVytah.StepName:='115 - Automaticky Rezim - kontrolujem paletku a zvoleny typ paletky pre aktualny model,vyplnam udaje paletky';
			SC_VstupVytah.IdleTime.PT:= T#200ms;
			SC_VstupVytah.AlarmTime.PT:= T#10s;

			IF Linka.PAR.Zvoleny_TypPaletky = RFID_Hlava_1.PAR.PrecitanyTypPaletky THEN
				Paletka[i].CisloPaletky:= RFID_Hlava_1.PAR.PrecitaneCisloPaletky;
				Paletka[i].TypPaletky:= Linka.PAR.Zvoleny_TypPaletky;
				Paletka[i].NazovModelu:= Linka.PAR.Zvoleny_MODEL;
				Paletka[i].CisloLOT:= Linka.PAR.Zvoleny_LOT;
				Paletka[i].Robot_CisloProgramu:= Linka.PAR.Zvolene_CisloProgramuRobota;
				Paletka[i].Kamera_CisloProgramu_QRkod:= Linka.PAR.Zvolene_KamCisloProg_QRkod;
				Paletka[i].Kamera_CisloProgramu_DMkod:= Linka.PAR.Zvolene_KamCisloProg_DMkod;
				Paletka[i].NazovPaletky:= '';
				brsstrcat(ADR(Paletka[i].NazovPaletky),ADR(Paletka[i].CisloPaletky));
				brsstrcat(ADR(Paletka[i].NazovPaletky),ADR('_'));
				brsstrcat(ADR(Paletka[i].NazovPaletky),ADR(Paletka[i].TypPaletky));
				Paletka[i].ReturnProcessName:= '';
				Paletka[i].TypVyroby:= '';
				Paletka[i].StavPaletky:= 'OK';
				Paletka[i].Cistenie_DONE:= FALSE;
				Paletka[i].StavCistenia:= '';
				Paletka[i].NalepenieEtikety_DONE:= FALSE;
				Paletka[i].StavNalepeniaEtikety:= '';
				Paletka[i].InternySerialNumber:= '';
				Paletka[i].ZakaznickeCislo:= '';
				Paletka[i].PrecitaneZnakyZakaznickehoDMkodu:= '';
				Paletka[i].StavCitania_InternehoQRkodu:= '';
				Paletka[i].StavCitania_ZakaznickehoDMkodu:= '';
				Paletka[i].StavCitania_KontrolaZnakov:= '';
				Paletka[i].StavKontrolyBielehoPaternu:= '';
				Paletka[i].StavPorovnaniaDMkoduZoServerom:= '';
				Paletka[i].StavKomunikacie_DONE:= FALSE;
				SC_VstupVytah.ResetStep:= TRUE;
				SC_VstupVytah.Step:= 120;
			ELSIF Linka.Rezim_Priechodny THEN
				Paletka[i].StavPaletky:= 'PR';
				SC_VstupVytah.ResetStep:= TRUE;
				SC_VstupVytah.Step:= 120;
			ELSE
				SC_VstupVytah.ResetStep:= TRUE;
				SC_VstupVytah.Step:= 118;
			END_IF

		118:
			SC_VstupVytah.StepName:='118 - Automaticky Rezim - cakam na vymenu zlej paletky a potvrdenie bannerom';
			SC_VstupVytah.IdleTime.PT:= T#2s;
			SC_VstupVytah.AlarmTime.PT:= T#10s;

			Vizu.ZobrazHlasenie_NespravTypPaletky:= 0;

			IF NOT Blikac500ms THEN
				VstupVytah.OUT.Banner_CervenaLED_IOS1:= TRUE;
				VstupVytah.OUT.Banner_ZelenaLED_IOS1:= TRUE;
			ELSE
				VstupVytah.OUT.Banner_ZelenaLED_IOS1:= FALSE;
				VstupVytah.OUT.Banner_CervenaLED_IOS1:= FALSE;
			END_IF

			IF VstupVytah.KoniecCyklu THEN
				SC_VstupVytah.ResetStep:= TRUE;
				SC_VstupVytah.Step:= 0;
			ELSIF Safety.STAV.BarieraVstupVytahu_AKTIVNA AND VstupVytah.IN.BannerPotvrdeny_IOS1 THEN
				VstupVytah.OUT.Banner_CervenaLED_IOS1:= FALSE;
				VstupVytah.OUT.Banner_ZelenaLED_IOS1:= FALSE;
				Vizu.ZobrazHlasenie_NespravTypPaletky:= 1;
				SC_VstupVytah.ResetStep:= TRUE;
				SC_VstupVytah.Step:= 100;
			ELSIF Safety.STAV.BarieraVstupVytahu_AKTIVNA AND NOT VstupVytah.IN.PritomnostPaletky_IS3 THEN
				VstupVytah.OUT.Banner_CervenaLED_IOS1:= FALSE;
				VstupVytah.OUT.Banner_ZelenaLED_IOS1:= FALSE;
				Vizu.ZobrazHlasenie_NespravTypPaletky:= 1;
				SC_VstupVytah.ResetStep:= TRUE;
				SC_VstupVytah.Step:= 100;
			END_IF

		120:
			SC_VstupVytah.StepName:='120 - Automaticky Rezim - cakam na vlozenie kusu a potvrdenie banerom alebo aktivnu barieru vstupneho vytahu a vyvezenie na stoper pred cistenim';
			SC_VstupVytah.IdleTime.PT:= T#2s;
			SC_VstupVytah.AlarmTime.PT:= T#10s;

			SC_VstupVytah.IdleTime.IN:= VstupVytah.IN.PritomnostPaletky_IS3 AND (VstupVytah.IN.PritomnostProduktu_OS2 OR Linka.Rezim_Priechodny) AND Safety.STAV.BarieraVstupVytahu_AKTIVNA;

			IF VstupVytah.IN.BannerPotvrdeny_IOS1 AND NOT Linka.Rezim_Priechodny AND VstupVytah.IN.PritomnostProduktu_OS2 AND Safety.STAV.BarieraVstupVytahu_AKTIVNA THEN
				VstupVytah.STAV.ObsluhaPotvrdilaBanner:= TRUE;
			ELSIF VstupVytah.IN.BannerPotvrdeny_IOS1 AND Linka.Rezim_Priechodny AND NOT VstupVytah.IN.PritomnostProduktu_OS2 AND Safety.STAV.BarieraVstupVytahu_AKTIVNA THEN
				VstupVytah.STAV.ObsluhaPotvrdilaBanner:= TRUE;
			END_IF

			IF VstupVytah.STAV.ObsluhaPotvrdilaBanner THEN
				VstupVytah.OUT.Banner_ZelenaLED_IOS1:= FALSE;
				VstupVytah.OUT.Banner_CervenaLED_IOS1:= TRUE;
			ELSE
				VstupVytah.OUT.Banner_CervenaLED_IOS1:= FALSE;
				VstupVytah.OUT.Banner_ZelenaLED_IOS1:= TRUE;
			END_IF

			IF VstupVytah.KoniecCyklu THEN
				SC_VstupVytah.ResetStep:= TRUE;
				SC_VstupVytah.Step:= 0;
			ELSIF Linka.Rezim_Priechodny AND VstupVytah.IN.PritomnostPaletky_IS3 AND NOT VstupVytah.IN.PritomnostProduktu_OS2 AND Safety.STAV.BarieraVstupVytahu_AKTIVNA AND VstupVytah.STAV.ObsluhaPotvrdilaBanner AND StoperPredCistenim.STAV.PoINIT AND NOT StoperPredCistenim.IN.PritomnostPaletky_IS4 AND NOT StoperPredCistenim.OUT.StoperZASUN_YV005 THEN
				VstupVytah.STAV.ObsluhaPotvrdilaBanner:= FALSE;
				SC_VstupVytah.ResetStep:= TRUE;
				SC_VstupVytah.Step:= 130;
			ELSIF Linka.Rezim_Priechodny AND VstupVytah.IN.PritomnostPaletky_IS3 AND NOT VstupVytah.IN.PritomnostProduktu_OS2 AND NOT VstupVytah_Banner_AKTIVNY AND SC_VstupVytah.IdleTime.Q AND StoperPredCistenim.STAV.PoINIT AND NOT StoperPredCistenim.IN.PritomnostPaletky_IS4 AND NOT StoperPredCistenim.OUT.StoperZASUN_YV005 THEN
				VstupVytah.OUT.Banner_ZelenaLED_IOS1:= FALSE;
				VstupVytah.OUT.Banner_CervenaLED_IOS1:= TRUE;
				VstupVytah.STAV.ObsluhaPotvrdilaBanner:= FALSE;
				SC_VstupVytah.ResetStep:= TRUE;
				SC_VstupVytah.Step:= 130;
			ELSIF NOT Linka.Rezim_Priechodny AND VstupVytah.IN.PritomnostPaletky_IS3 AND VstupVytah.IN.PritomnostProduktu_OS2 AND Safety.STAV.BarieraVstupVytahu_AKTIVNA AND VstupVytah.STAV.ObsluhaPotvrdilaBanner AND StoperPredCistenim.STAV.PoINIT AND NOT StoperPredCistenim.IN.PritomnostPaletky_IS4 AND NOT StoperPredCistenim.OUT.StoperZASUN_YV005 THEN
				VstupVytah.STAV.ObsluhaPotvrdilaBanner:= FALSE;
				SC_VstupVytah.ResetStep:= TRUE;
				SC_VstupVytah.Step:= 130;
			ELSIF NOT Linka.Rezim_Priechodny AND VstupVytah.IN.PritomnostPaletky_IS3 AND VstupVytah.IN.PritomnostProduktu_OS2 AND NOT VstupVytah_Banner_AKTIVNY AND SC_VstupVytah.IdleTime.Q AND StoperPredCistenim.STAV.PoINIT AND NOT StoperPredCistenim.IN.PritomnostPaletky_IS4 AND NOT StoperPredCistenim.OUT.StoperZASUN_YV005 THEN
				VstupVytah.OUT.Banner_ZelenaLED_IOS1:= FALSE;
				VstupVytah.OUT.Banner_CervenaLED_IOS1:= TRUE;
				VstupVytah.STAV.ObsluhaPotvrdilaBanner:= FALSE;
				SC_VstupVytah.ResetStep:= TRUE;
				SC_VstupVytah.Step:= 130;
			ELSIF NOT VstupVytah.IN.PritomnostPaletky_IS3 AND Safety.STAV.BarieraVstupVytahu_AKTIVNA THEN
				VstupVytah.STAV.ObsluhaPotvrdilaBanner:= FALSE;
				VstupVytah.OUT.Banner_ZelenaLED_IOS1:= FALSE;
				VstupVytah.OUT.Banner_CervenaLED_IOS1:= FALSE;
				SC_VstupVytah.ResetStep:= TRUE;
				SC_VstupVytah.Step:= 112;
			END_IF

		130:
			SC_VstupVytah.StepName:='130 - Automaticky Rezim - otvorenie dveri vytahu';
			SC_VstupVytah.IdleTime.PT:= T#500ms;
			SC_VstupVytah.AlarmTime.PT:= T#1s;

			SC_VstupVytah.AlarmTime.IN:= NOT Safety.STAV.BarieraVstupVytahu_AKTIVNA;

			IF NOT SC_VstupVytah.Switch1 THEN
				Dvere_OTVOR:= TRUE;
				SC_VstupVytah.Switch1:= TRUE;
			END_IF

			IF VstupVytah.IN.DvereVytahuOtvorene_MS1 THEN
				SC_VstupVytah.ResetStep:= TRUE;
				SC_VstupVytah.Step:= 138;
			ELSIF SC_VstupVytah.AlarmTime.Q THEN
				Alarmy[46]:= TRUE;
				PoruchaVstupnehoVytahu:= TRUE;
				SC_VstupVytah.ResetStep:= TRUE;
				SC_VstupVytah.Step:= 0;
			END_IF

		138:
			SC_VstupVytah.StepName:='125 - Automaticky Rezim - vyvezenie paletky na stoper pred cistenim';
			SC_VstupVytah.IdleTime.PT:= T#500ms;
			SC_VstupVytah.AlarmTime.PT:= T#10s;

			IF NOT SC_VstupVytah.Switch1 THEN
				VstupVytah.OUT.Dopravnik_ChodVPRED_ELR1:= TRUE;
				SC_VstupVytah.AlarmTime.IN:= TRUE;
				VstupVytah.STAV.PrebiehaVyvazaniePaletky:= TRUE;
				VstupnyVytah_Statistika.IN.START_MeraniaCasu:= TRUE;
				VstupnyVytah_Statistika.IN.ZAPIS_MeraniaCasu:= TRUE;
				SC_VstupVytah.Switch1:= TRUE;
			END_IF

			IF NOT VstupVytah.IN.PritomnostPaletky_IS3 AND NOT VstupVytah.IN.PrechodDopravnikaVytahu_OS1 AND StoperPredCistenim.IN.PritomnostPaletky_IS4 THEN
				VstupVytah.OUT.Dopravnik_ChodVPRED_ELR1:= FALSE;
				VstupVytah.STAV.PrebiehaVyvazaniePaletky:= FALSE;
				VstupVytah.OUT.Banner_CervenaLED_IOS1:= FALSE;
				SC_VstupVytah.ResetStep:= TRUE;
				SC_VstupVytah.Step:= 140;
			ELSIF NOT Safety.STAV.BarieraVstupVytahu_AKTIVNA THEN
				Alarmy[46]:= TRUE;
				PoruchaVstupnehoVytahu:= TRUE;
				SC_VstupVytah.ResetStep:= TRUE;
				SC_VstupVytah.Step:= 0;
			ELSIF SC_VstupVytah.AlarmTime.Q THEN
				Alarmy[48]:= TRUE;
				PoruchaVstupnehoVytahu:= TRUE;
				SC_VstupVytah.ResetStep:= TRUE;
				SC_VstupVytah.Step:= 0;
			END_IF

		140:
			SC_VstupVytah.StepName:='140 - Automaticky Rezim - zatvorenie dveri vytahu';
			SC_VstupVytah.IdleTime.PT:= T#500ms;
			SC_VstupVytah.AlarmTime.PT:= T#10s;

			IF NOT SC_VstupVytah.Switch1 THEN
				Dvere_ZATVOR:= TRUE;
				SC_VstupVytah.Switch1:= TRUE;
			END_IF

			IF VstupVytah.IN.DvereVytahuZatvorene_MS2 THEN
				VstupVytah.STAV.ObsluhaPotvrdilaBanner:= FALSE;
				VstupVytah.OUT.Banner_ZelenaLED_IOS1:= FALSE;
				SC_VstupVytah.ResetStep:= TRUE;
				SC_VstupVytah.Step:= 100;
			ELSIF NOT Safety.STAV.BarieraVstupVytahu_AKTIVNA THEN
				Alarmy[46]:= TRUE;
				PoruchaVstupnehoVytahu:= TRUE;
				SC_VstupVytah.ResetStep:= TRUE;
				SC_VstupVytah.Step:= 0;
			END_IF

			//*******************************************************Manuálny režim*******************************************************************************//
		700:
			SC_VstupVytah.StepName:='700 - Manualny Rezim';
			SC_VstupVytah.IdleTime.PT:= T#8s;
			SC_VstupVytah.AlarmTime.PT:= T#5s;

			//Ovládanie dopravníka//
			IF VstupVytah.RR_Dopravnik_VPRED THEN
				VstupVytah.OUT.Dopravnik_ChodVZAD_ELR1:= FALSE;
				VstupVytah.OUT.Dopravnik_ChodVPRED_ELR1:= TRUE;
			ELSIF VstupVytah.RR_Dopravnik_VZAD THEN
				VstupVytah.OUT.Dopravnik_ChodVPRED_ELR1:= FALSE;
				VstupVytah.OUT.Dopravnik_ChodVZAD_ELR1:= TRUE;
			ELSE
				VstupVytah.OUT.Dopravnik_ChodVPRED_ELR1:= FALSE;
				VstupVytah.OUT.Dopravnik_ChodVZAD_ELR1:= FALSE;
			END_IF

	END_CASE

				END_PROGRAM

PROGRAM _EXIT
				(* Insert code here *)

				END_PROGRAM
```

#### Variables.var - Local variables
```iecst
VAR
	SC_OvlMenica : SequenceControlTyp := (0);
	Zdvih_JoggHORE : BOOL := FALSE;
	Zdvih_JoggDOLE : BOOL := FALSE;
	Zdvih_POLOHUJ : BOOL := FALSE;
	Zdvih_HOME : BOOL := FALSE;
	SC_OvlDveri : SequenceControlTyp := (0);
	Dvere_OTVOR : BOOL := FALSE;
	Dvere_ZATVOR : BOOL := FALSE;
	i : USINT := 0;
	VstupnePoleUSINT : ARRAY[1..20] OF USINT;
	VystupnePoleStringov : ARRAY[1..20] OF STRING[80];
	h : USINT := 0;
	PocetZnakovUDINT : UDINT;
	PocetZnakovUSINT : USINT;
	g : USINT := 0;
	AktualNacitanyZnak : USINT;
END_VAR
```

#### OvlMenica.st
```iecst
ACTION OvlMenica:

	//Otáčka motora = zdvih 10 mm//

	//CANopen adresa meniča - 34//

	//Volanie funkčného bloku//
	VstupVytah.MenicZdvihu_FM2();

	//Volanie funkcie SequenceControl//
	SequenceControl(SC:= SC_OvlMenica);

	//Prepnutie meniča do stavu READY//
	IF EDGEPOS(Safety.STAV.SafetyPLC_Nabehlo)THEN
		IF NOT VstupVytah.MenicZdvihu_FM2.STAV.READY THEN
			VstupVytah.MenicZdvihu_FM2.CMD.Potvrd_PORUCHU:= TRUE;
		END_IF
	ELSIF EDGEPOS(Safety.STAV.ZonaVstupnyVytah_AKTIVNA)THEN
		IF NOT VstupVytah.MenicZdvihu_FM2.STAV.READY THEN
			VstupVytah.MenicZdvihu_FM2.CMD.Potvrd_PORUCHU:= TRUE;
		END_IF
	END_IF

	//Parametre meniča//
	VstupVytah.MenicZdvihu_FM2.PAR.TypKomunikacieProfinet:= 0;
	VstupVytah.MenicZdvihu_FM2.PAR.ZadanaPozicia_MM:= (VstupVytah.PAR.Zdvih_ZadanaPozicia * 100);
	VstupVytah.STAV.Zdvih_AktualnaPozicia:= (VstupVytah.MenicZdvihu_FM2.PAR.AktualnaPozicia_MM/100);
	VstupVytah.STAV.Zdvih_AktualnaRychlost:= VstupVytah.MenicZdvihu_FM2.PAR.AktualnaFrekvencia_Hz;
	VstupVytah.STAV.Zdvih_HomingOK:= VstupVytah.MenicZdvihu_FM2.STAV.Homing_OK;
	VstupVytah.STAV.Zdvih_PoziciaDosiahnuta:= VstupVytah.MenicZdvihu_FM2.STAV.Pozicia_DOSIAHNUTA;
	VstupVytah.STAV.Zdvih_BUSY:= VstupVytah.MenicZdvihu_FM2.STAV.RUN;

	//Preposielanie IO meniča cez komunikáciu//
	VstupVytah.IN.ReferencnySnimacZdvihu:= VstupVytah.MenicZdvihu_FM2.PAR.BUS_OUT_Bit_0;
	VstupVytah.IN.HornyLimitZdvihu:= VstupVytah.MenicZdvihu_FM2.PAR.BUS_OUT_Bit_1;
	VstupVytah.MenicZdvihu_FM2.PAR.BUS_IN_Bit_0:= VstupVytah.IN.SpodnyLimitZdvihu;

	IF Zdvih_HOME THEN
		VstupVytah.IN.SpodnyLimitZdvihu:= TRUE;
	ELSE
		VstupVytah.IN.SpodnyLimitZdvihu:= NOT VstupVytah.IN.ReferencnySnimacZdvihu;
	END_IF

	IF NOT Safety.STAV.ZonaVstupnyVytah_AKTIVNA THEN
		SC_OvlMenica.Step:= 0;
	END_IF

	CASE SC_OvlMenica.Step OF

		0:
			SC_OvlMenica.StepName:= '0 - Nulovanie';
			Zdvih_JoggHORE:= FALSE;
			Zdvih_JoggDOLE:= FALSE;
			Zdvih_POLOHUJ:= FALSE;
			Zdvih_HOME:= FALSE;
			VstupVytah.MenicZdvihu_FM2.CMD.HOME:= FALSE;
			VstupVytah.MenicZdvihu_FM2.CMD.Chod_VPRED:= FALSE;
			VstupVytah.MenicZdvihu_FM2.CMD.Chod_VZAD:= FALSE;
			VstupVytah.MenicZdvihu_FM2.CMD.Polohuj:= FALSE;
			VstupVytah.STAV.Homing_BUSY:= FALSE;

			IF SC_VstupVytah.Step <> 0 AND VstupVytah.MenicZdvihu_FM2.STAV.READY AND NOT VstupVytah.MenicZdvihu_FM2.STAV.PORUCHA AND Safety.STAV.ZonaVstupnyVytah_AKTIVNA THEN
				SC_OvlMenica.ResetStep:= TRUE;
				SC_OvlMenica.Step:= 1;
			END_IF

		1:
			SC_OvlMenica.StepName:= '1 - Rozhodnutie o cinnosti';
			IF Zdvih_JoggHORE THEN
				SC_OvlMenica.Step:= 10;
			ELSIF Zdvih_JoggDOLE THEN
				SC_OvlMenica.Step:= 20;
			ELSIF Zdvih_HOME THEN
				SC_OvlMenica.Step:= 30;
			ELSIF Zdvih_POLOHUJ THEN
				SC_OvlMenica.Step:= 40;
			END_IF

		10:
			SC_OvlMenica.StepName:= '10 - Jogg HORE';
			SC_OvlMenica.IdleTime.PT:= T#3s;
			SC_OvlMenica.AlarmTime.PT:= T#3s;

			VstupVytah.MenicZdvihu_FM2.PAR.ZadanaFrekvencia_Hz:= VstupVytah.PAR.Zdvih_ZadanaJoggRychlost;

			IF NOT SC_OvlMenica.Switch1 AND VstupVytah.IN.HornyLimitZdvihu THEN
				VstupVytah.MenicZdvihu_FM2.CMD.Chod_VPRED:= TRUE;
				SC_OvlMenica.Switch1:= TRUE;
			END_IF

			IF NOT Zdvih_JoggHORE THEN
				SC_OvlMenica.ResetStep:= TRUE;
				SC_OvlMenica.Step:= 0;
			ELSIF NOT VstupVytah.IN.HornyLimitZdvihu THEN
				SC_OvlMenica.ResetStep:= TRUE;
				SC_OvlMenica.Step:= 0;
			END_IF

		20:
			SC_OvlMenica.StepName:= '20 - Jogg DOLE';
			SC_OvlMenica.IdleTime.PT:= T#3s;
			SC_OvlMenica.AlarmTime.PT:= T#3s;

			VstupVytah.MenicZdvihu_FM2.PAR.ZadanaFrekvencia_Hz:= VstupVytah.PAR.Zdvih_ZadanaJoggRychlost;

			IF NOT SC_OvlMenica.Switch1 AND VstupVytah.IN.SpodnyLimitZdvihu THEN
				VstupVytah.MenicZdvihu_FM2.CMD.Chod_VZAD:= TRUE;
				SC_OvlMenica.Switch1:= TRUE;
			END_IF

			IF NOT Zdvih_JoggDOLE THEN
				SC_OvlMenica.ResetStep:= TRUE;
				SC_OvlMenica.Step:= 0;
			ELSIF NOT VstupVytah.IN.SpodnyLimitZdvihu THEN
				SC_OvlMenica.ResetStep:= TRUE;
				SC_OvlMenica.Step:= 0;
			END_IF

		30:
			SC_OvlMenica.StepName:= '30 - Homing - kontrola referencneho snimaca';
			SC_OvlMenica.IdleTime.PT:= T#500ms;
			SC_OvlMenica.AlarmTime.PT:= T#3s;

			VstupVytah.STAV.Homing_BUSY:= TRUE;

			IF VstupVytah.IN.ReferencnySnimacZdvihu THEN
				SC_OvlMenica.ResetStep:= TRUE;
				SC_OvlMenica.Step:= 31;
			ELSE
				SC_OvlMenica.ResetStep:= TRUE;
				SC_OvlMenica.Step:= 32;
			END_IF

		31:
			SC_OvlMenica.StepName:= '31 - Homing - presun vytahu nad referencny snimac';
			SC_OvlMenica.IdleTime.PT:= T#1s;
			SC_OvlMenica.AlarmTime.PT:= T#2s;

			SC_OvlMenica.IdleTime.IN:= NOT VstupVytah.IN.ReferencnySnimacZdvihu;

			IF NOT SC_OvlMenica.Switch1 THEN
				VstupVytah.MenicZdvihu_FM2.CMD.Chod_VPRED:= TRUE;
				SC_OvlMenica.Switch1:= TRUE;
			END_IF

			IF SC_OvlMenica.IdleTime.Q THEN
				VstupVytah.MenicZdvihu_FM2.CMD.Chod_VPRED:= FALSE;
				SC_OvlMenica.AlarmTime.IN:= TRUE;
			END_IF

			IF SC_OvlMenica.AlarmTime.Q THEN
				SC_OvlMenica.ResetStep:= TRUE;
				SC_OvlMenica.Step:= 32;
			END_IF

		32:
			SC_OvlMenica.StepName:= '32 - Homing - spustenie homingu';
			SC_OvlMenica.IdleTime.PT:= T#500ms;
			SC_OvlMenica.AlarmTime.PT:= T#3s;

			IF NOT SC_OvlMenica.Switch1 THEN
				VstupVytah.MenicZdvihu_FM2.CMD.HOME:= TRUE;
				SC_OvlMenica.IdleTime.IN:= TRUE;
				SC_OvlMenica.Switch1:= TRUE;
			END_IF

			IF VstupVytah.STAV.Zdvih_HomingOK AND SC_OvlMenica.IdleTime.Q THEN
				SC_OvlMenica.ResetStep:= TRUE;
				SC_OvlMenica.Step:= 0;
			ELSIF NOT Zdvih_HOME THEN
				SC_OvlMenica.ResetStep:= TRUE;
				SC_OvlMenica.Step:= 0;
			END_IF

		40:
			SC_OvlMenica.StepName:= '40 - Polohovanie';
			SC_OvlMenica.IdleTime.PT:= T#1s;
			SC_OvlMenica.AlarmTime.PT:= T#3s;

			VstupVytah.MenicZdvihu_FM2.PAR.ZadanaFrekvencia_Hz:= VstupVytah.PAR.Zdvih_ZadanaRychlost;

			IF NOT SC_OvlMenica.Switch1 THEN
				VstupVytah.MenicZdvihu_FM2.CMD.Polohuj:= TRUE;
				SC_OvlMenica.IdleTime.IN:= TRUE;
				SC_OvlMenica.Switch1:= TRUE;
			END_IF

			IF (*(VstupVytah.STAV.Zdvih_AktualnaPozicia = VstupVytah.PAR.Zdvih_ZadanaPozicia) AND*) SC_OvlMenica.IdleTime.Q AND VstupVytah.STAV.Zdvih_PoziciaDosiahnuta THEN
				VstupVytah.STAV.VytahNapolohovany:= TRUE;
				SC_OvlMenica.ResetStep:= TRUE;
				SC_OvlMenica.Step:= 0;
			ELSIF NOT Zdvih_POLOHUJ THEN
				SC_OvlMenica.ResetStep:= TRUE;
				SC_OvlMenica.Step:= 0;
			END_IF

	END_CASE

END_ACTION
```

#### OvlDveri.st
```iecst
ACTION OvlDveri:

	//Volanie funkcie SequenceControl//
	SequenceControl(SC:= SC_OvlDveri);

	CASE SC_OvlDveri.Step OF

		0:
			SC_OvlDveri.StepName:= '0 - Nulovanie';
			Dvere_OTVOR:= FALSE;
			Dvere_ZATVOR:= FALSE;
			VstupVytah.OUT.DvereVytahu_OTVOR_YV002:= FALSE;
			VstupVytah.OUT.DvereVytahu_ZATVOR_YV001:= FALSE;

			IF SC_VstupVytah.Step <> 0 THEN
				SC_OvlDveri.ResetStep:= TRUE;
				SC_OvlDveri.Step:= 1;
			END_IF

		1:
			SC_OvlDveri.StepName:= '1 - Rozhodnutie o cinnosti';
			IF Dvere_OTVOR THEN
				SC_OvlDveri.Step:= 10;
			ELSIF Dvere_ZATVOR THEN
				SC_OvlDveri.Step:= 20;
			END_IF

		10:
			SC_OvlDveri.StepName:= '10 - Otvorenie dveri';
			SC_OvlDveri.IdleTime.PT:= T#3s;
			SC_OvlDveri.AlarmTime.PT:= T#6s;

			IF VstupVytah.Automat THEN
				SC_OvlDveri.AlarmTime.IN:= TRUE;
			ELSE
				SC_OvlDveri.IdleTime.IN:= TRUE;
			END_IF

			IF NOT SC_OvlDveri.Switch1 THEN
				VstupVytah.OUT.DvereVytahu_ZATVOR_YV001:= FALSE;
				VstupVytah.OUT.DvereVytahu_OTVOR_YV002:= TRUE;
				SC_OvlDveri.Switch1:= TRUE;
			END_IF

			IF VstupVytah.IN.DvereVytahuOtvorene_MS1 OR SC_OvlDveri.IdleTime.Q THEN
				SC_OvlDveri.ResetStep:= TRUE;
				SC_OvlDveri.Step:= 0;
			ELSIF NOT Safety.STAV.BarieraVstupVytahu_AKTIVNA THEN
				SC_OvlDveri.ResetStep:= TRUE;
				SC_OvlDveri.Step:= 0;
			ELSIF SC_OvlDveri.AlarmTime.Q THEN
				Alarmy[42]:= TRUE;
				PoruchaVstupnehoVytahu:= TRUE;
				SC_OvlDveri.ResetStep:= TRUE;
				SC_OvlDveri.Step:= 0;
			END_IF

		20:
			SC_OvlDveri.StepName:= '20 - Zatvorenie dveri';
			SC_OvlDveri.IdleTime.PT:= T#3s;
			SC_OvlDveri.AlarmTime.PT:= T#6s;

			IF VstupVytah.Automat THEN
				SC_OvlDveri.AlarmTime.IN:= TRUE;
			ELSE
				SC_OvlDveri.IdleTime.IN:= TRUE;
			END_IF

			IF NOT SC_OvlDveri.Switch1 THEN
				VstupVytah.OUT.DvereVytahu_OTVOR_YV002:= FALSE;
				VstupVytah.OUT.DvereVytahu_ZATVOR_YV001:= TRUE;
				SC_OvlDveri.Switch1:= TRUE;
			END_IF

			IF VstupVytah.IN.DvereVytahuZatvorene_MS2 OR SC_OvlDveri.IdleTime.Q THEN
				SC_OvlDveri.ResetStep:= TRUE;
				SC_OvlDveri.Step:= 0;
			ELSIF NOT Safety.STAV.BarieraVstupVytahu_AKTIVNA THEN
				SC_OvlDveri.ResetStep:= TRUE;
				SC_OvlDveri.Step:= 0;
			ELSIF SC_OvlDveri.AlarmTime.Q THEN
				Alarmy[43]:= TRUE;
				PoruchaVstupnehoVytahu:= TRUE;
				SC_OvlDveri.ResetStep:= TRUE;
				SC_OvlDveri.Step:= 0;
			END_IF

	END_CASE

END_ACTION
```

#### OvlCitackyRFID.st
```iecst
ACTION OvlCitackyRFID:

	//***********************************************************************Riadenie RFID hlavy 1 - Vstupny výťah**********************************************************************//

	//Volanie funkcie SequenceControl//
	SequenceControl(SC:= SC_Hlava_1);

	//*************************Komunikácia*******************************//
	//INPUTS//
	RFID_Hlava_1.STAV.PritomnostCipu:= RFID_Hlava_1.IN.BYTE_IN[0].0;
	RFID_Hlava_1.IN.Bit_CP:= RFID_Hlava_1.IN.BYTE_IN[0].0;
	RFID_Hlava_1.IN.Bit_AA:= RFID_Hlava_1.IN.BYTE_IN[0].1;
	RFID_Hlava_1.IN.Bit_AE:= RFID_Hlava_1.IN.BYTE_IN[0].2;
	RFID_Hlava_1.IN.Bit_AF:= RFID_Hlava_1.IN.BYTE_IN[0].3;
	RFID_Hlava_1.IN.Bit_MT:= RFID_Hlava_1.IN.BYTE_IN[0].4;
	RFID_Hlava_1.IN.Bit_TO:= RFID_Hlava_1.IN.BYTE_IN[0].5;
	RFID_Hlava_1.IN.Bit_HF:= RFID_Hlava_1.IN.BYTE_IN[0].6;
	RFID_Hlava_1.IN.Bit_BB:= RFID_Hlava_1.IN.BYTE_IN[0].7;

	//OUTPUTS//
	RFID_Hlava_1.OUT.BYTE_OUT[0].0:= RFID_Hlava_1.OUT.Bit_AV;
	RFID_Hlava_1.OUT.BYTE_OUT[31].0:= RFID_Hlava_1.OUT.Bit_AV;
	RFID_Hlava_1.OUT.BYTE_OUT[0].2:= RFID_Hlava_1.OUT.Bit_GR;
	RFID_Hlava_1.OUT.BYTE_OUT[31].2:= RFID_Hlava_1.OUT.Bit_GR;
	RFID_Hlava_1.OUT.BYTE_OUT[0].5:= RFID_Hlava_1.OUT.Bit_KA;
	RFID_Hlava_1.OUT.BYTE_OUT[31].5:= RFID_Hlava_1.OUT.Bit_KA;
	RFID_Hlava_1.OUT.BYTE_OUT[0].6:= RFID_Hlava_1.OUT.Bit_TI;
	RFID_Hlava_1.OUT.BYTE_OUT[31].6:= RFID_Hlava_1.OUT.Bit_TI;

	//Prečítané znaky//
	RFID_Hlava_1.PAR.PrecitaneCisloPaletky_POLE[0]:= RFID_Hlava_1.IN.BYTE_IN[1];
	RFID_Hlava_1.PAR.PrecitaneCisloPaletky_POLE[1]:= RFID_Hlava_1.IN.BYTE_IN[2];
	RFID_Hlava_1.PAR.PrecitaneCisloPaletky_POLE[2]:= RFID_Hlava_1.IN.BYTE_IN[3];
	RFID_Hlava_1.PAR.PrecitaneCisloPaletky_POLE[3]:= RFID_Hlava_1.IN.BYTE_IN[4];
	RFID_Hlava_1.PAR.PrecitaneCisloPaletky_POLE[4]:= RFID_Hlava_1.IN.BYTE_IN[5];
	RFID_Hlava_1.PAR.PrecitaneCisloPaletky_POLE[5]:= RFID_Hlava_1.IN.BYTE_IN[6];
	RFID_Hlava_1.PAR.PrecitaneCisloPaletky_POLE[6]:= RFID_Hlava_1.IN.BYTE_IN[7];
	RFID_Hlava_1.PAR.PrecitaneCisloPaletky_POLE[7]:= RFID_Hlava_1.IN.BYTE_IN[8];
	RFID_Hlava_1.PAR.PrecitaneCisloPaletky_POLE[8]:= RFID_Hlava_1.IN.BYTE_IN[9];
	RFID_Hlava_1.PAR.PrecitaneCisloPaletky_POLE[9]:= RFID_Hlava_1.IN.BYTE_IN[10];

	brsmemcpy(ADR(RFID_Hlava_1.PAR.Precitane_Cislo_Typ_Paletky),ADR(RFID_Hlava_1.PAR.PrecitaneCisloPaletky_POLE),SIZEOF(RFID_Hlava_1.PAR.PrecitaneCisloPaletky_POLE));

	//Rozdelenie prečítanej správy na číslo paletky a model//
	IF RFID_Hlava_1.STAV.PritomnostCipu THEN
		brsmemset(ADR(VstupnePoleUSINT),0,SIZEOF(VstupnePoleUSINT)); //Vymazanie vstupneho pola
		brsmemset(ADR(VystupnePoleStringov),0,SIZEOF(VystupnePoleStringov)); //Vymazanie výstupneho pola znakov
		PocetZnakovUDINT := brsstrlen(ADR(RFID_Hlava_1.PAR.Precitane_Cislo_Typ_Paletky)); //Zistenie počtu znakov vstupnej spravy
		PocetZnakovUSINT:= UDINT_TO_USINT(PocetZnakovUDINT);
		brsmemcpy(ADR(VstupnePoleUSINT),ADR(RFID_Hlava_1.PAR.Precitane_Cislo_Typ_Paletky),SIZEOF(RFID_Hlava_1.PAR.Precitane_Cislo_Typ_Paletky)); //Vyplnenie polia znakmy vstupnej správy
		h:= 1;
		FOR g:= 1 TO PocetZnakovUSINT BY 1 DO
			IF VstupnePoleUSINT[g] <> 59 THEN //59 je oddelovací znak bodkočiarka
				AktualNacitanyZnak:= VstupnePoleUSINT[g];
				brsstrcat(ADR(VystupnePoleStringov[h]),ADR(AktualNacitanyZnak));
			ELSE
				h:= h + 1;
			END_IF
		END_FOR
		RFID_Hlava_1.PAR.PrecitaneCisloPaletky:= VystupnePoleStringov[1];
		RFID_Hlava_1.PAR.PrecitanyTypPaletky:= VystupnePoleStringov[2];
	ELSE
		RFID_Hlava_1.PAR.PrecitaneCisloPaletky:= '';
		RFID_Hlava_1.PAR.PrecitanyTypPaletky:= '';
	END_IF

	CASE SC_Hlava_1.Step OF

		0:
			SC_Hlava_1.StepName:= '0 - Nulovanie';
			RFID_Hlava_1.CMD.CitajDATA:= FALSE;
			RFID_Hlava_1.CMD.ZapisDATA:= FALSE;
			RFID_Hlava_1.CMD.CitaciuHlavu_VYPNI:= FALSE;
			RFID_Hlava_1.OUT.Bit_AV:= FALSE;
			RFID_Hlava_1.OUT.Bit_GR:= FALSE;
			RFID_Hlava_1.OUT.Bit_TI:= FALSE;
			RFID_Hlava_1.OUT.Bit_KA:= FALSE;

			IF RFID_Hlava_1.STAV.PritomnostCipu THEN
				SC_Hlava_1.ResetStep:= TRUE;
				SC_Hlava_1.Step:= 1;
			END_IF

		1:
			SC_Hlava_1.StepName:= '1 - Rozhodnutie o cinnosti';
			IF NOT RFID_Hlava_1.STAV.PritomnostCipu THEN
				SC_Hlava_1.Step:= 0;
			ELSIF RFID_Hlava_1.CMD.CitajDATA THEN
				RFID_Hlava_1.STAV.CitanieDat_OK:= FALSE;
				RFID_Hlava_1.STAV.CitanieDat_ERROR:= FALSE;
				SC_Hlava_1.Step:= 10;
			ELSIF RFID_Hlava_1.CMD.ZapisDATA THEN
				RFID_Hlava_1.STAV.ZapisDat_OK:= FALSE;
				RFID_Hlava_1.STAV.ZapisDat_ERROR:= FALSE;
				SC_Hlava_1.Step:= 20;
			ELSIF RFID_Hlava_1.CMD.CitaciuHlavu_VYPNI THEN
				SC_Hlava_1.Step:= 30;
			END_IF

		10:
			SC_Hlava_1.StepName:= '10 - Citanie dat';
			SC_Hlava_1.IdleTime.PT:= T#3s;
			SC_Hlava_1.AlarmTime.PT:= T#6s;

			RFID_Hlava_1.IN.Old_Bit_TO:= RFID_Hlava_1.IN.Bit_TO;
			RFID_Hlava_1.OUT.BYTE_OUT[1]:= 1; //Kommand - 1 - čítanie, 2 - zápis
			RFID_Hlava_1.OUT.BYTE_OUT[2]:= 0; //Štartovacia adresa čítania (LSB) - na 2 byte začína zapisovať načítané znaky
			RFID_Hlava_1.OUT.BYTE_OUT[3]:= 0; //Štartovacia adresa čítania (HSB)
			RFID_Hlava_1.OUT.BYTE_OUT[4]:= 10; //Počet bajtov čítania (LSB) - 10 znakov
			RFID_Hlava_1.OUT.BYTE_OUT[5]:= 0; //Počet bajtov čítania (HSB)
			RFID_Hlava_1.OUT.Bit_AV:= TRUE;

			SC_Hlava_1.ResetStep:= TRUE;
			SC_Hlava_1.Step:= 11;

		11:
			SC_Hlava_1.StepName:= '11 - Citanie dat';
			SC_Hlava_1.IdleTime.PT:= T#3s;
			SC_Hlava_1.AlarmTime.PT:= T#2s;

			IF RFID_Hlava_1.IN.Bit_AA AND RFID_Hlava_1.IN.Bit_AE AND (RFID_Hlava_1.IN.Old_Bit_TO <> RFID_Hlava_1.IN.Bit_TO) THEN
				RFID_Hlava_1.STAV.CitanieDat_OK:= TRUE;
				SC_Hlava_1.ResetStep:= TRUE;
				SC_Hlava_1.Step:= 12;
			ELSIF RFID_Hlava_1.IN.Bit_AF THEN
				RFID_Hlava_1.STAV.CitanieDat_ERROR:= TRUE;
				SC_Hlava_1.ResetStep:= TRUE;
				SC_Hlava_1.Step:= 12;
			END_IF

		12:
			SC_Hlava_1.StepName:= '12 - Citanie dat';
			SC_Hlava_1.IdleTime.PT:= T#3s;
			SC_Hlava_1.AlarmTime.PT:= T#6s;

			RFID_Hlava_1.OUT.Bit_AV:= FALSE;

			IF NOT RFID_Hlava_1.IN.Bit_AA AND NOT RFID_Hlava_1.IN.Bit_AE AND NOT RFID_Hlava_1.IN.Bit_AF THEN
				SC_Hlava_1.ResetStep:= TRUE;
				SC_Hlava_1.Step:= 0;
			END_IF

		20:
			SC_Hlava_1.StepName:= '20 - Zápis dat';
			SC_Hlava_1.IdleTime.PT:= T#3s;
			SC_Hlava_1.AlarmTime.PT:= T#6s;

			RFID_Hlava_1.IN.Old_Bit_TO:= RFID_Hlava_1.IN.Bit_TO;
			RFID_Hlava_1.OUT.BYTE_OUT[1]:= 2; //Kommand - 1 - čítanie, 2 - zápis
			RFID_Hlava_1.OUT.BYTE_OUT[2]:= 0; //Štartovacia adresa zápisu (LSB) - na 2 byte začína zapisovať znaky
			RFID_Hlava_1.OUT.BYTE_OUT[3]:= 0; //Štartovacia adresa zápisu (HSB)
			RFID_Hlava_1.OUT.BYTE_OUT[4]:= 10; //Počet bajtov zápisu (LSB) - 10 znakov
			RFID_Hlava_1.OUT.BYTE_OUT[5]:= 0; //Počet bajtov zápisu (HSB)
			RFID_Hlava_1.OUT.Bit_AV:= TRUE;

			SC_Hlava_1.ResetStep:= TRUE;
			SC_Hlava_1.Step:= 21;

		21:
			SC_Hlava_1.StepName:= '21 - Zápis dat';
			SC_Hlava_1.IdleTime.PT:= T#3s;
			SC_Hlava_1.AlarmTime.PT:= T#2s;

			IF RFID_Hlava_1.IN.Bit_AA AND (RFID_Hlava_1.IN.Old_Bit_TO <> RFID_Hlava_1.IN.Bit_TO) THEN
				SC_Hlava_1.ResetStep:= TRUE;
				SC_Hlava_1.Step:= 22;
			END_IF

		22:
			SC_Hlava_1.StepName:= '21 - Zápis dat';
			SC_Hlava_1.IdleTime.PT:= T#3s;
			SC_Hlava_1.AlarmTime.PT:= T#6s;

			brsstrcpy(ADR(RFID_Hlava_1.PAR.ZadaneCisloPaletky_POLE),ADR(RFID_Hlava_1.PAR.Zadane_Cislo_Typ_Paletky));
			RFID_Hlava_1.OUT.BYTE_OUT[1]:= RFID_Hlava_1.PAR.ZadaneCisloPaletky_POLE[0];
			RFID_Hlava_1.OUT.BYTE_OUT[2]:= RFID_Hlava_1.PAR.ZadaneCisloPaletky_POLE[1];
			RFID_Hlava_1.OUT.BYTE_OUT[3]:= RFID_Hlava_1.PAR.ZadaneCisloPaletky_POLE[2];
			RFID_Hlava_1.OUT.BYTE_OUT[4]:= RFID_Hlava_1.PAR.ZadaneCisloPaletky_POLE[3];
			RFID_Hlava_1.OUT.BYTE_OUT[5]:= RFID_Hlava_1.PAR.ZadaneCisloPaletky_POLE[4];
			RFID_Hlava_1.OUT.BYTE_OUT[6]:= RFID_Hlava_1.PAR.ZadaneCisloPaletky_POLE[5];
			RFID_Hlava_1.OUT.BYTE_OUT[7]:= RFID_Hlava_1.PAR.ZadaneCisloPaletky_POLE[6];
			RFID_Hlava_1.OUT.BYTE_OUT[8]:= RFID_Hlava_1.PAR.ZadaneCisloPaletky_POLE[7];
			RFID_Hlava_1.OUT.BYTE_OUT[9]:= RFID_Hlava_1.PAR.ZadaneCisloPaletky_POLE[8];
			RFID_Hlava_1.OUT.BYTE_OUT[10]:= RFID_Hlava_1.PAR.ZadaneCisloPaletky_POLE[9];

			IF RFID_Hlava_1.OUT.Bit_TI THEN
				RFID_Hlava_1.OUT.Bit_TI:= FALSE;
				SC_Hlava_1.ResetStep:= TRUE;
				SC_Hlava_1.Step:= 23;
			ELSE
				RFID_Hlava_1.OUT.Bit_TI:= TRUE;
				SC_Hlava_1.ResetStep:= TRUE;
				SC_Hlava_1.Step:= 23;
			END_IF

		23:
			SC_Hlava_1.StepName:= '23 - Zápis dat';
			SC_Hlava_1.IdleTime.PT:= T#3s;
			SC_Hlava_1.AlarmTime.PT:= T#2s;

			IF RFID_Hlava_1.IN.Bit_AE THEN
				RFID_Hlava_1.STAV.ZapisDat_OK:= TRUE;
				SC_Hlava_1.ResetStep:= TRUE;
				SC_Hlava_1.Step:= 24;
			ELSIF RFID_Hlava_1.IN.Bit_AF THEN
				RFID_Hlava_1.STAV.ZapisDat_ERROR:= TRUE;
				SC_Hlava_1.ResetStep:= TRUE;
				SC_Hlava_1.Step:= 24;
			END_IF

		24:
			SC_Hlava_1.StepName:= '22 - Zápis dat';
			SC_Hlava_1.IdleTime.PT:= T#3s;
			SC_Hlava_1.AlarmTime.PT:= T#6s;

			RFID_Hlava_1.OUT.Bit_AV:= FALSE;

			IF NOT RFID_Hlava_1.IN.Bit_AA AND NOT RFID_Hlava_1.IN.Bit_AE AND NOT RFID_Hlava_1.IN.Bit_AF THEN
				SC_Hlava_1.ResetStep:= TRUE;
				SC_Hlava_1.Step:= 0;
			END_IF

		30:
			SC_Hlava_1.StepName:= '30 - Vypnutie citacej hlavy';
			SC_Hlava_1.IdleTime.PT:= T#3s;
			SC_Hlava_1.AlarmTime.PT:= T#2s;

			RFID_Hlava_1.OUT.Bit_KA:= TRUE;

			IF NOT RFID_Hlava_1.CMD.CitaciuHlavu_VYPNI THEN
				SC_Hlava_1.ResetStep:= TRUE;
				SC_Hlava_1.Step:= 0;
			END_IF

	END_CASE

END_ACTION
```

### Program Logical/Program/StoperPredCistenim (IEC)

#### Main.st - Init, cyclic, exit code
```iecst
PROGRAM _INIT
	(* Insert code here *)

END_PROGRAM

PROGRAM _CYCLIC

	//Volanie funkcie SequenceControl//
	SequenceControl(SC:= SC_StoperPredCistenim);

	//Volanie podprogramov//
	OvlCitackyRFID;

	//Reset sekcie //
	IF StoperPredCistenim.Reset THEN
		SC_StoperPredCistenim.Step:= 0;
		StoperPredCistenim.Reset:= FALSE;
	ELSIF NOT Safety.STAV.ZonaCS_AKTIVNA THEN
		SC_StoperPredCistenim.Step:= 0;
	END_IF

	CASE SC_StoperPredCistenim.Step OF

		0:
			SC_StoperPredCistenim.StepName:='0 - Nulovanie';
			StoperPredCistenim.Automat:= FALSE;
			StoperPredCistenim.KoniecCyklu:= FALSE;
			StoperPredCistenim.Manual:= FALSE;
			StoperPredCistenim.STAV.PoINIT:= FALSE;
			StoperPredCistenim.OUT.StoperZASUN_YV005:= FALSE;
			StoperPredCistenim.STAV.PrebiehaVyvazaniePaletky:= FALSE;
			Linka.OUT.IonJednotka_START:= FALSE;
			Linka.STAV.IonizacnaJednotka_BUSY:= FALSE;
			StoperPredCistenim_Statistika.IN.START_MeraniaCasu:= FALSE;

			IF Safety.STAV.ZonaCS_AKTIVNA AND Linka.IN.TlakVzduchu_OK_S2 AND NOT NastalaPorucha AND Linka.STAV.Hardware_OK THEN
				SC_StoperPredCistenim.ResetStep:= TRUE;
				SC_StoperPredCistenim.Step:= 1;
			END_IF

		1:
			SC_StoperPredCistenim.StepName:='1 - Cakam na spustenie vyroby';
			StoperPredCistenim.KoniecCyklu:= FALSE;
			IF StoperPredCistenim.Automat THEN
				SC_StoperPredCistenim.Step:= 2;
			ELSIF StoperPredCistenim.Manual THEN
				SC_StoperPredCistenim.Step:= 700;
			END_IF

			//********************************************************Inicializácia****************************************************************************//
		2:
			SC_StoperPredCistenim.StepName:='2 - Inicializacia - cakam na spustenie inicializacie';
			SC_StoperPredCistenim.IdleTime.PT:= T#4s;
			SC_StoperPredCistenim.AlarmTime.PT:= T#5s;

			IF DopravCistenia.STAV.PoINIT THEN
				SC_StoperPredCistenim.ResetStep:= TRUE;
				SC_StoperPredCistenim.Step:= 3;
			END_IF

		3:
			SC_StoperPredCistenim.StepName:='3 - Inicializacia - hladanie paletky';
			SC_StoperPredCistenim.IdleTime.PT:= T#5s;
			SC_StoperPredCistenim.AlarmTime.PT:= T#5s;
			SC_StoperPredCistenim.IdleTime.IN:= TRUE;

			IF StoperPredCistenim.IN.PritomnostPaletky_IS4 THEN
				StoperPredCistenim.STAV.PoINIT:= TRUE;
				SC_StoperPredCistenim.ResetStep:= TRUE;
				SC_StoperPredCistenim.Step:= 101;
			ELSIF SC_StoperPredCistenim.IdleTime.Q THEN
				StoperPredCistenim.STAV.PoINIT:= TRUE;
				SC_StoperPredCistenim.ResetStep:= TRUE;
				SC_StoperPredCistenim.Step:= 100;
			END_IF

			//********************************************************Automatický režim****************************************************************************//
		100:
			SC_StoperPredCistenim.StepName:='100 - Automaticky Rezim - cakam na príchod paletky na stoper';
			SC_StoperPredCistenim.IdleTime.PT:= T#200ms;
			SC_StoperPredCistenim.AlarmTime.PT:= T#30s;

			SC_StoperPredCistenim.AlarmTime.IN:= TRUE;

			IF SC_StoperPredCistenim.AlarmTime.Q THEN
				Linka.OUT.IonJednotka_START:= FALSE;
				Linka.STAV.IonizacnaJednotka_BUSY:= FALSE;
			END_IF

			DopravCistenia.PAR.ZadanaRychlost:= 50;

			SC_StoperPredCistenim.IdleTime.IN:= StoperPredCistenim.IN.PritomnostPaletky_IS4;

			IF StoperPredCistenim.KoniecCyklu THEN
				SC_StoperPredCistenim.ResetStep:= TRUE;
				SC_StoperPredCistenim.Step:= 0;
			ELSIF SC_StoperPredCistenim.IdleTime.Q THEN
				StoperPredCistenim_Statistika.IN.START_MeraniaCasu:= TRUE;
				StoperPredCistenim_Statistika.IN.ZAPIS_MeraniaCasu:= TRUE;
				SC_StoperPredCistenim.ResetStep:= TRUE;
				SC_StoperPredCistenim.Step:= 101;
			END_IF

		101:
			SC_StoperPredCistenim.StepName:='101 - Automaticky Rezim - cakam na vyvezenie paletky na stoper za cistenim';
			SC_StoperPredCistenim.IdleTime.PT:= T#200ms;
			SC_StoperPredCistenim.AlarmTime.PT:= T#30s;

			SC_StoperPredCistenim.AlarmTime.IN:= TRUE;

			IF SC_StoperPredCistenim.AlarmTime.Q THEN
				Linka.OUT.IonJednotka_START:= FALSE;
				Linka.STAV.IonizacnaJednotka_BUSY:= FALSE;
			END_IF

			IF StoperPredCistenim.KoniecCyklu THEN
				SC_StoperPredCistenim.ResetStep:= TRUE;
				SC_StoperPredCistenim.Step:= 0;
			ELSIF SC_StoperPoCisteni.Step = 100 AND (NOT StoperPoCisteni.IN.PritomnostPaletky_IS6 OR NOT StoperPoCisteni.IN.ZaplnenieBuffera_IS5) AND NOT StoperPoCisteni.STAV.PrebiehaVyvazaniePaletky THEN
				IF Linka.Rezim_BezCistenia THEN
					SC_StoperPredCistenim.ResetStep:= TRUE;
					SC_StoperPredCistenim.Step:= 105;
				ELSIF Linka.Rezim_Priechodny THEN
					SC_StoperPredCistenim.ResetStep:= TRUE;
					SC_StoperPredCistenim.Step:= 105;
				ELSE
					SC_StoperPredCistenim.ResetStep:= TRUE;
					SC_StoperPredCistenim.Step:= 103;
				END_IF
			ELSIF StoperPoCisteni.STAV.PoINIT AND NOT StoperPoCisteni.IN.ZaplnenieBuffera_IS5 THEN
				IF Linka.Rezim_BezCistenia THEN
					SC_StoperPredCistenim.ResetStep:= TRUE;
					SC_StoperPredCistenim.Step:= 105;
				ELSIF Linka.Rezim_Priechodny THEN
					SC_StoperPredCistenim.ResetStep:= TRUE;
					SC_StoperPredCistenim.Step:= 105;
				ELSE
					SC_StoperPredCistenim.ResetStep:= TRUE;
					SC_StoperPredCistenim.Step:= 103;
				END_IF
			END_IF

		103:
			SC_StoperPredCistenim.StepName:='103 - Automaticky Rezim - cakam na spustenie cistenia';
			SC_StoperPredCistenim.IdleTime.PT:= T#2s;
			SC_StoperPredCistenim.AlarmTime.PT:= T#10s;

			DopravCistenia.PAR.ZadanaRychlost:= Linka.PAR.Zvolena_RychlostDopravPriCisteni;

			IF NOT SC_StoperPredCistenim.Switch1 THEN
				Linka.OUT.IonJednotka_START:= TRUE;
				SC_StoperPredCistenim.IdleTime.IN:= TRUE;
				SC_StoperPredCistenim.Switch1:= TRUE;
			END_IF

			IF NOT Linka.STAV.PoruchaOtacaniaTrysiek AND SC_StoperPredCistenim.IdleTime.Q THEN
				Linka.STAV.IonizacnaJednotka_BUSY:= TRUE;
				SC_StoperPredCistenim.ResetStep:= TRUE;
				SC_StoperPredCistenim.Step:= 105;
			ELSIF Linka.STAV.IonizacnaJednotka_BUSY THEN
				SC_StoperPredCistenim.ResetStep:= TRUE;
				SC_StoperPredCistenim.Step:= 105;
			ELSIF Linka.STAV.PoruchaOtacaniaTrysiek THEN
				PoruchaCistenia:= TRUE;
				SC_StoperPredCistenim.ResetStep:= TRUE;
				SC_StoperPredCistenim.Step:= 0;
			END_IF

		105:
			SC_StoperPredCistenim.StepName:='105 - Automaticky Rezim - vyvazam paletku na RFID snimac po cisteni, zastavenie cistenia';
			SC_StoperPredCistenim.IdleTime.PT:= T#200ms;
			SC_StoperPredCistenim.AlarmTime.PT:= T#10s;

			SC_StoperPredCistenim.IdleTime.IN:= NOT StoperPredCistenim.IN.PritomnostPaletky_IS4;

			IF NOT SC_StoperPredCistenim.Switch1 THEN
				StoperPredCistenim.OUT.StoperZASUN_YV005:= TRUE;
				SC_StoperPredCistenim.AlarmTime.IN:= TRUE;
				StoperPredCistenim.STAV.PrebiehaVyvazaniePaletky:= TRUE;
				SC_StoperPredCistenim.Switch1:= TRUE;
			END_IF

			IF SC_StoperPredCistenim.IdleTime.Q THEN
				StoperPredCistenim.OUT.StoperZASUN_YV005:= FALSE;
				SC_StoperPredCistenim.AlarmTime.IN:= FALSE;
			END_IF

			IF NOT StoperPredCistenim.OUT.StoperZASUN_YV005 AND RFID_Hlava_4.STAV.PritomnostCipu THEN
				(*Linka.OUT.IonJednotka_START:= FALSE;*)
				SC_StoperPredCistenim.ResetStep:= TRUE;
				SC_StoperPredCistenim.Step:= 107;
			END_IF

		107:
			SC_StoperPredCistenim.StepName:='107 - Automaticky Rezim - precitanie cisla paletky';
			SC_StoperPredCistenim.IdleTime.PT:= T#20ms;
			SC_StoperPredCistenim.AlarmTime.PT:= T#10s;

			SC_StoperPredCistenim.AlarmTime.IN:= TRUE;

			SC_StoperPredCistenim.IdleTime.IN:= RFID_Hlava_4.STAV.PritomnostCipu;

			IF RFID_Hlava_4.PAR.PrecitaneCisloPaletky <> '' THEN
				i:=  STRING_TO_USINT(RFID_Hlava_4.PAR.PrecitaneCisloPaletky);
				SC_StoperPredCistenim.ResetStep:= TRUE;
				SC_StoperPredCistenim.Step:= 110;
			END_IF

			IF SC_StoperPredCistenim.AlarmTime.Q THEN
				Alarmy[70]:= TRUE;
				PoruchaCistenia:= TRUE;
				SC_StoperPredCistenim.ResetStep:= TRUE;
				SC_StoperPredCistenim.Step:= 0;
			END_IF

		110:
			SC_StoperPredCistenim.StepName:='110 - Automaticky Rezim - zapis stavu cistenia na paletku';
			SC_StoperPredCistenim.IdleTime.PT:= T#200ms;
			SC_StoperPredCistenim.AlarmTime.PT:= T#10s;

			IF Linka.Rezim_BezCistenia THEN
				Paletka[i].Cistenie_DONE:= TRUE;
				Paletka[i].StavCistenia:= 'OK';
				Paletka[i].StavPaletky:= 'OK';
				SC_StoperPredCistenim.ResetStep:= TRUE;
				SC_StoperPredCistenim.Step:= 115;
			ELSIF Linka.Rezim_Priechodny THEN
				SC_StoperPredCistenim.ResetStep:= TRUE;
				SC_StoperPredCistenim.Step:= 115;
			ELSIF NOT Linka.STAV.PoruchaOtacaniaTrysiek THEN
				Paletka[i].Cistenie_DONE:= TRUE;
				Paletka[i].StavCistenia:= 'OK';
				Paletka[i].StavPaletky:= 'OK';
				SC_StoperPredCistenim.ResetStep:= TRUE;
				SC_StoperPredCistenim.Step:= 115;
			ELSIF Linka.STAV.PoruchaOtacaniaTrysiek THEN
				Paletka[i].Cistenie_DONE:= TRUE;
				Paletka[i].StavCistenia:= 'NG';
				Paletka[i].StavPaletky:= 'NG';
				SC_StoperPredCistenim.ResetStep:= TRUE;
				SC_StoperPredCistenim.Step:= 115;
			END_IF

		115:
			SC_StoperPredCistenim.StepName:='115 - Automaticky Rezim - vyvazam paletku na stoper po cisteni';
			SC_StoperPredCistenim.IdleTime.PT:= T#4s;
			SC_StoperPredCistenim.AlarmTime.PT:= T#10s;

			DopravCistenia.PAR.ZadanaRychlost:= 80;

			IF NOT SC_StoperPredCistenim.Switch1 THEN
				DopravCistenia.Dopravnik_RUN:= TRUE;
				SC_StoperPredCistenim.Switch1:= TRUE;
			END_IF

			IF StoperPoCisteni.IN.PritomnostPaletky_IS6 THEN
				StoperPredCistenim.STAV.PrebiehaVyvazaniePaletky:= FALSE;
				IF NOT Linka.STAV.PoruchaOtacaniaTrysiek THEN
					SC_StoperPredCistenim.ResetStep:= TRUE;
					SC_StoperPredCistenim.Step:= 100;
				ELSE
					PoruchaCistenia:= TRUE;
					SC_StoperPredCistenim.ResetStep:= TRUE;
					SC_StoperPredCistenim.Step:= 0;
				END_IF
			END_IF

			//*******************************************************Manuálny režim*******************************************************************************//
		700:
			SC_StoperPredCistenim.StepName:='700 - Manualny Rezim';
			SC_StoperPredCistenim.IdleTime.PT:= T#8s;
			SC_StoperPredCistenim.AlarmTime.PT:= T#5s;

	END_CASE

END_PROGRAM

PROGRAM _EXIT
	(* Insert code here *)

END_PROGRAM
```

#### Variables.var - Local variables
```iecst
VAR
	VstupnePoleUSINT : ARRAY[1..20] OF USINT;
	VystupnePoleStringov : ARRAY[1..20] OF STRING[80];
	h : USINT := 0;
	PocetZnakovUDINT : UDINT;
	PocetZnakovUSINT : USINT;
	g : USINT := 0;
	AktualNacitanyZnak : USINT;
	i : USINT := 0;
END_VAR
```

#### OvlCitackyRFID.st
```iecst
ACTION OvlCitackyRFID:

	//***********************************************************************Riadenie RFID hlavy 1 - Vstupny výťah**********************************************************************//

	//Volanie funkcie SequenceControl//
	SequenceControl(SC:= SC_Hlava_4);

	//*************************Komunikácia*******************************//
	//INPUTS//
	RFID_Hlava_4.STAV.PritomnostCipu:= RFID_Hlava_4.IN.BYTE_IN[0].0;
	RFID_Hlava_4.IN.Bit_CP:= RFID_Hlava_4.IN.BYTE_IN[0].0;
	RFID_Hlava_4.IN.Bit_AA:= RFID_Hlava_4.IN.BYTE_IN[0].1;
	RFID_Hlava_4.IN.Bit_AE:= RFID_Hlava_4.IN.BYTE_IN[0].2;
	RFID_Hlava_4.IN.Bit_AF:= RFID_Hlava_4.IN.BYTE_IN[0].3;
	RFID_Hlava_4.IN.Bit_MT:= RFID_Hlava_4.IN.BYTE_IN[0].4;
	RFID_Hlava_4.IN.Bit_TO:= RFID_Hlava_4.IN.BYTE_IN[0].5;
	RFID_Hlava_4.IN.Bit_HF:= RFID_Hlava_4.IN.BYTE_IN[0].6;
	RFID_Hlava_4.IN.Bit_BB:= RFID_Hlava_4.IN.BYTE_IN[0].7;

	//OUTPUTS//
	RFID_Hlava_4.OUT.BYTE_OUT[0].0:= RFID_Hlava_4.OUT.Bit_AV;
	RFID_Hlava_4.OUT.BYTE_OUT[31].0:= RFID_Hlava_4.OUT.Bit_AV;
	RFID_Hlava_4.OUT.BYTE_OUT[0].2:= RFID_Hlava_4.OUT.Bit_GR;
	RFID_Hlava_4.OUT.BYTE_OUT[31].2:= RFID_Hlava_4.OUT.Bit_GR;
	RFID_Hlava_4.OUT.BYTE_OUT[0].5:= RFID_Hlava_4.OUT.Bit_KA;
	RFID_Hlava_4.OUT.BYTE_OUT[31].5:= RFID_Hlava_4.OUT.Bit_KA;
	RFID_Hlava_4.OUT.BYTE_OUT[0].6:= RFID_Hlava_4.OUT.Bit_TI;
	RFID_Hlava_4.OUT.BYTE_OUT[31].6:= RFID_Hlava_4.OUT.Bit_TI;

	//Prečítané znaky//
	RFID_Hlava_4.PAR.PrecitaneCisloPaletky_POLE[0]:= RFID_Hlava_4.IN.BYTE_IN[1];
	RFID_Hlava_4.PAR.PrecitaneCisloPaletky_POLE[1]:= RFID_Hlava_4.IN.BYTE_IN[2];
	RFID_Hlava_4.PAR.PrecitaneCisloPaletky_POLE[2]:= RFID_Hlava_4.IN.BYTE_IN[3];
	RFID_Hlava_4.PAR.PrecitaneCisloPaletky_POLE[3]:= RFID_Hlava_4.IN.BYTE_IN[4];
	RFID_Hlava_4.PAR.PrecitaneCisloPaletky_POLE[4]:= RFID_Hlava_4.IN.BYTE_IN[5];
	RFID_Hlava_4.PAR.PrecitaneCisloPaletky_POLE[5]:= RFID_Hlava_4.IN.BYTE_IN[6];
	RFID_Hlava_4.PAR.PrecitaneCisloPaletky_POLE[6]:= RFID_Hlava_4.IN.BYTE_IN[7];
	RFID_Hlava_4.PAR.PrecitaneCisloPaletky_POLE[7]:= RFID_Hlava_4.IN.BYTE_IN[8];
	RFID_Hlava_4.PAR.PrecitaneCisloPaletky_POLE[8]:= RFID_Hlava_4.IN.BYTE_IN[9];
	RFID_Hlava_4.PAR.PrecitaneCisloPaletky_POLE[9]:= RFID_Hlava_4.IN.BYTE_IN[10];

	brsmemcpy(ADR(RFID_Hlava_4.PAR.Precitane_Cislo_Typ_Paletky),ADR(RFID_Hlava_4.PAR.PrecitaneCisloPaletky_POLE),SIZEOF(RFID_Hlava_4.PAR.PrecitaneCisloPaletky_POLE));

	//Rozdelenie prečítanej správy na číslo paletky a model//
	IF RFID_Hlava_4.STAV.PritomnostCipu THEN
		brsmemset(ADR(VstupnePoleUSINT),0,SIZEOF(VstupnePoleUSINT)); //Vymazanie vstupneho pola
		brsmemset(ADR(VystupnePoleStringov),0,SIZEOF(VystupnePoleStringov)); //Vymazanie výstupneho pola znakov
		PocetZnakovUDINT := brsstrlen(ADR(RFID_Hlava_4.PAR.Precitane_Cislo_Typ_Paletky)); //Zistenie počtu znakov vstupnej spravy
		PocetZnakovUSINT:= UDINT_TO_USINT(PocetZnakovUDINT);
		brsmemcpy(ADR(VstupnePoleUSINT),ADR(RFID_Hlava_4.PAR.Precitane_Cislo_Typ_Paletky),SIZEOF(RFID_Hlava_4.PAR.Precitane_Cislo_Typ_Paletky)); //Vyplnenie polia znakmy vstupnej správy
		h:= 1;
		FOR g:= 1 TO PocetZnakovUSINT BY 1 DO
			IF VstupnePoleUSINT[g] <> 59 THEN //59 je oddelovací znak bodkočiarka
				AktualNacitanyZnak:= VstupnePoleUSINT[g];
				brsstrcat(ADR(VystupnePoleStringov[h]),ADR(AktualNacitanyZnak));
			ELSE
				h:= h + 1;
			END_IF
		END_FOR
		RFID_Hlava_4.PAR.PrecitaneCisloPaletky:= VystupnePoleStringov[1];
		RFID_Hlava_4.PAR.PrecitanyTypPaletky:= VystupnePoleStringov[2];
	ELSE
		RFID_Hlava_4.PAR.PrecitaneCisloPaletky:= '';
		RFID_Hlava_4.PAR.PrecitanyTypPaletky:= '';
	END_IF

	CASE SC_Hlava_4.Step OF

		0:
			SC_Hlava_4.StepName:= '0 - Nulovanie';
			RFID_Hlava_4.CMD.CitajDATA:= FALSE;
			RFID_Hlava_4.CMD.ZapisDATA:= FALSE;
			RFID_Hlava_4.CMD.CitaciuHlavu_VYPNI:= FALSE;
			RFID_Hlava_4.OUT.Bit_AV:= FALSE;
			RFID_Hlava_4.OUT.Bit_GR:= FALSE;
			RFID_Hlava_4.OUT.Bit_TI:= FALSE;
			RFID_Hlava_4.OUT.Bit_KA:= FALSE;

			IF RFID_Hlava_4.STAV.PritomnostCipu THEN
				SC_Hlava_4.ResetStep:= TRUE;
				SC_Hlava_4.Step:= 1;
			END_IF

		1:
			SC_Hlava_4.StepName:= '1 - Rozhodnutie o cinnosti';
			IF NOT RFID_Hlava_4.STAV.PritomnostCipu THEN
				SC_Hlava_4.Step:= 0;
			ELSIF RFID_Hlava_4.CMD.CitajDATA THEN
				RFID_Hlava_4.STAV.CitanieDat_OK:= FALSE;
				RFID_Hlava_4.STAV.CitanieDat_ERROR:= FALSE;
				SC_Hlava_4.Step:= 10;
			ELSIF RFID_Hlava_4.CMD.ZapisDATA THEN
				RFID_Hlava_4.STAV.ZapisDat_OK:= FALSE;
				RFID_Hlava_4.STAV.ZapisDat_ERROR:= FALSE;
				SC_Hlava_4.Step:= 20;
			ELSIF RFID_Hlava_4.CMD.CitaciuHlavu_VYPNI THEN
				SC_Hlava_4.Step:= 30;
			END_IF

		10:
			SC_Hlava_4.StepName:= '10 - Citanie dat';
			SC_Hlava_4.IdleTime.PT:= T#3s;
			SC_Hlava_4.AlarmTime.PT:= T#6s;

			RFID_Hlava_4.IN.Old_Bit_TO:= RFID_Hlava_4.IN.Bit_TO;
			RFID_Hlava_4.OUT.BYTE_OUT[1]:= 1; //Kommand - 1 - čítanie, 2 - zápis
			RFID_Hlava_4.OUT.BYTE_OUT[2]:= 0; //Štartovacia adresa čítania (LSB) - na 2 byte začína zapisovať načítané znaky
			RFID_Hlava_4.OUT.BYTE_OUT[3]:= 0; //Štartovacia adresa čítania (HSB)
			RFID_Hlava_4.OUT.BYTE_OUT[4]:= 10; //Počet bajtov čítania (LSB) - 10 znakov
			RFID_Hlava_4.OUT.BYTE_OUT[5]:= 0; //Počet bajtov čítania (HSB)
			RFID_Hlava_4.OUT.Bit_AV:= TRUE;

			SC_Hlava_4.ResetStep:= TRUE;
			SC_Hlava_4.Step:= 11;

		11:
			SC_Hlava_4.StepName:= '11 - Citanie dat';
			SC_Hlava_4.IdleTime.PT:= T#3s;
			SC_Hlava_4.AlarmTime.PT:= T#2s;

			IF RFID_Hlava_4.IN.Bit_AA AND RFID_Hlava_4.IN.Bit_AE AND (RFID_Hlava_4.IN.Old_Bit_TO <> RFID_Hlava_4.IN.Bit_TO) THEN
				RFID_Hlava_4.STAV.CitanieDat_OK:= TRUE;
				SC_Hlava_4.ResetStep:= TRUE;
				SC_Hlava_4.Step:= 12;
			ELSIF RFID_Hlava_4.IN.Bit_AF THEN
				RFID_Hlava_4.STAV.CitanieDat_ERROR:= TRUE;
				SC_Hlava_4.ResetStep:= TRUE;
				SC_Hlava_4.Step:= 12;
			END_IF

		12:
			SC_Hlava_4.StepName:= '12 - Citanie dat';
			SC_Hlava_4.IdleTime.PT:= T#3s;
			SC_Hlava_4.AlarmTime.PT:= T#6s;

			RFID_Hlava_4.OUT.Bit_AV:= FALSE;

			IF NOT RFID_Hlava_4.IN.Bit_AA AND NOT RFID_Hlava_4.IN.Bit_AE AND NOT RFID_Hlava_4.IN.Bit_AF THEN
				SC_Hlava_4.ResetStep:= TRUE;
				SC_Hlava_4.Step:= 0;
			END_IF

		20:
			SC_Hlava_4.StepName:= '20 - Zápis dat';
			SC_Hlava_4.IdleTime.PT:= T#3s;
			SC_Hlava_4.AlarmTime.PT:= T#6s;

			RFID_Hlava_4.IN.Old_Bit_TO:= RFID_Hlava_4.IN.Bit_TO;
			RFID_Hlava_4.OUT.BYTE_OUT[1]:= 2; //Kommand - 1 - čítanie, 2 - zápis
			RFID_Hlava_4.OUT.BYTE_OUT[2]:= 0; //Štartovacia adresa zápisu (LSB) - na 2 byte začína zapisovať znaky
			RFID_Hlava_4.OUT.BYTE_OUT[3]:= 0; //Štartovacia adresa zápisu (HSB)
			RFID_Hlava_4.OUT.BYTE_OUT[4]:= 10; //Počet bajtov zápisu (LSB) - 10 znakov
			RFID_Hlava_4.OUT.BYTE_OUT[5]:= 0; //Počet bajtov zápisu (HSB)
			RFID_Hlava_4.OUT.Bit_AV:= TRUE;

			SC_Hlava_4.ResetStep:= TRUE;
			SC_Hlava_4.Step:= 21;

		21:
			SC_Hlava_4.StepName:= '21 - Zápis dat';
			SC_Hlava_4.IdleTime.PT:= T#3s;
			SC_Hlava_4.AlarmTime.PT:= T#2s;

			IF RFID_Hlava_4.IN.Bit_AA AND (RFID_Hlava_4.IN.Old_Bit_TO <> RFID_Hlava_4.IN.Bit_TO) THEN
				SC_Hlava_4.ResetStep:= TRUE;
				SC_Hlava_4.Step:= 22;
			END_IF

		22:
			SC_Hlava_4.StepName:= '21 - Zápis dat';
			SC_Hlava_4.IdleTime.PT:= T#3s;
			SC_Hlava_4.AlarmTime.PT:= T#6s;

			brsstrcpy(ADR(RFID_Hlava_4.PAR.ZadaneCisloPaletky_POLE),ADR(RFID_Hlava_4.PAR.Zadane_Cislo_Typ_Paletky));
			RFID_Hlava_4.OUT.BYTE_OUT[1]:= RFID_Hlava_4.PAR.ZadaneCisloPaletky_POLE[0];
			RFID_Hlava_4.OUT.BYTE_OUT[2]:= RFID_Hlava_4.PAR.ZadaneCisloPaletky_POLE[1];
			RFID_Hlava_4.OUT.BYTE_OUT[3]:= RFID_Hlava_4.PAR.ZadaneCisloPaletky_POLE[2];
			RFID_Hlava_4.OUT.BYTE_OUT[4]:= RFID_Hlava_4.PAR.ZadaneCisloPaletky_POLE[3];
			RFID_Hlava_4.OUT.BYTE_OUT[5]:= RFID_Hlava_4.PAR.ZadaneCisloPaletky_POLE[4];
			RFID_Hlava_4.OUT.BYTE_OUT[6]:= RFID_Hlava_4.PAR.ZadaneCisloPaletky_POLE[5];
			RFID_Hlava_4.OUT.BYTE_OUT[7]:= RFID_Hlava_4.PAR.ZadaneCisloPaletky_POLE[6];
			RFID_Hlava_4.OUT.BYTE_OUT[8]:= RFID_Hlava_4.PAR.ZadaneCisloPaletky_POLE[7];
			RFID_Hlava_4.OUT.BYTE_OUT[9]:= RFID_Hlava_4.PAR.ZadaneCisloPaletky_POLE[8];
			RFID_Hlava_4.OUT.BYTE_OUT[10]:= RFID_Hlava_4.PAR.ZadaneCisloPaletky_POLE[9];

			IF RFID_Hlava_4.OUT.Bit_TI THEN
				RFID_Hlava_4.OUT.Bit_TI:= FALSE;
				SC_Hlava_4.ResetStep:= TRUE;
				SC_Hlava_4.Step:= 23;
			ELSE
				RFID_Hlava_4.OUT.Bit_TI:= TRUE;
				SC_Hlava_4.ResetStep:= TRUE;
				SC_Hlava_4.Step:= 23;
			END_IF

		23:
			SC_Hlava_4.StepName:= '23 - Zápis dat';
			SC_Hlava_4.IdleTime.PT:= T#3s;
			SC_Hlava_4.AlarmTime.PT:= T#2s;

			IF RFID_Hlava_4.IN.Bit_AE THEN
				RFID_Hlava_4.STAV.ZapisDat_OK:= TRUE;
				SC_Hlava_4.ResetStep:= TRUE;
				SC_Hlava_4.Step:= 24;
			ELSIF RFID_Hlava_4.IN.Bit_AF THEN
				RFID_Hlava_4.STAV.ZapisDat_ERROR:= TRUE;
				SC_Hlava_4.ResetStep:= TRUE;
				SC_Hlava_4.Step:= 24;
			END_IF

		24:
			SC_Hlava_4.StepName:= '22 - Zápis dat';
			SC_Hlava_4.IdleTime.PT:= T#3s;
			SC_Hlava_4.AlarmTime.PT:= T#6s;

			RFID_Hlava_4.OUT.Bit_AV:= FALSE;

			IF NOT RFID_Hlava_4.IN.Bit_AA AND NOT RFID_Hlava_4.IN.Bit_AE AND NOT RFID_Hlava_4.IN.Bit_AF THEN
				SC_Hlava_4.ResetStep:= TRUE;
				SC_Hlava_4.Step:= 0;
			END_IF

		30:
			SC_Hlava_4.StepName:= '30 - Vypnutie citacej hlavy';
			SC_Hlava_4.IdleTime.PT:= T#3s;
			SC_Hlava_4.AlarmTime.PT:= T#2s;

			RFID_Hlava_4.OUT.Bit_KA:= TRUE;

			IF NOT RFID_Hlava_4.CMD.CitaciuHlavu_VYPNI THEN
				SC_Hlava_4.ResetStep:= TRUE;
				SC_Hlava_4.Step:= 0;
			END_IF

	END_CASE

END_ACTION
```

### Program Logical/Program/StoperPoCisteni (IEC)

#### Main.st - Init, cyclic, exit code
```iecst
PROGRAM _INIT
	(* Insert code here *)

END_PROGRAM

PROGRAM _CYCLIC

	//Volanie funkcie SequenceControl//
	SequenceControl(SC:= SC_StoperPoCisteni);

	//Reset sekcie //
	IF StoperPoCisteni.Reset THEN
		SC_StoperPoCisteni.Step:= 0;
		StoperPoCisteni.Reset:= FALSE;
	ELSIF NOT Safety.STAV.ZonaCS_AKTIVNA THEN
		SC_StoperPoCisteni.Step:= 0;
	END_IF

	CASE SC_StoperPoCisteni.Step OF

		0:
			SC_StoperPoCisteni.StepName:='0 - Nulovanie';
			StoperPoCisteni.Automat:= FALSE;
			StoperPoCisteni.KoniecCyklu:= FALSE;
			StoperPoCisteni.Manual:= FALSE;
			StoperPoCisteni.STAV.PoINIT:= FALSE;
			StoperPoCisteni.OUT.StoperZASUN_YV006:= FALSE;
			StoperPoCisteni.STAV.PrebiehaVyvazaniePaletky:= FALSE;
			StoperPoCisteni_Statistika.IN.START_MeraniaCasu:= FALSE;

			IF Safety.STAV.ZonaCS_AKTIVNA AND Linka.IN.TlakVzduchu_OK_S2 AND NOT NastalaPorucha AND Linka.STAV.Hardware_OK THEN
				SC_StoperPoCisteni.ResetStep:= TRUE;
				SC_StoperPoCisteni.Step:= 1;
			END_IF

		1:
			SC_StoperPoCisteni.StepName:='1 - Cakam na spustenie vyroby';
			StoperPoCisteni.KoniecCyklu:= FALSE;
			IF StoperPoCisteni.Automat THEN
				SC_StoperPoCisteni.Step:= 2;
			ELSIF StoperPoCisteni.Manual THEN
				SC_StoperPoCisteni.Step:= 700;
			END_IF

			//********************************************************Inicializácia****************************************************************************//

		2:
			SC_StoperPoCisteni.StepName:='2 - Inicializacia - cakam na spustenie inicializacie';
			SC_StoperPoCisteni.IdleTime.PT:= T#4s;
			SC_StoperPoCisteni.AlarmTime.PT:= T#5s;

			IF DopravCistenia.STAV.PoINIT THEN
				SC_StoperPoCisteni.ResetStep:= TRUE;
				SC_StoperPoCisteni.Step:= 3;
			END_IF

		3:
			SC_StoperPoCisteni.StepName:='3 - Inicializacia - hladanie paletky';
			SC_StoperPoCisteni.IdleTime.PT:= T#5s;
			SC_StoperPoCisteni.AlarmTime.PT:= T#5s;
			SC_StoperPoCisteni.IdleTime.IN:= TRUE;

			IF StoperPoCisteni.IN.PritomnostPaletky_IS6 THEN
				StoperPoCisteni.STAV.PoINIT:= TRUE;
				SC_StoperPoCisteni.ResetStep:= TRUE;
				SC_StoperPoCisteni.Step:= 101;
			ELSIF SC_StoperPoCisteni.IdleTime.Q THEN
				StoperPoCisteni.STAV.PoINIT:= TRUE;
				SC_StoperPoCisteni.ResetStep:= TRUE;
				SC_StoperPoCisteni.Step:= 100;
			END_IF

			//********************************************************Automatický režim****************************************************************************//
		100:
			SC_StoperPoCisteni.StepName:='100 - Automaticky Rezim - cakam na príchod paletky na stoper';
			SC_StoperPoCisteni.IdleTime.PT:= T#200ms;
			SC_StoperPoCisteni.AlarmTime.PT:= T#5s;

			SC_StoperPoCisteni.IdleTime.IN:= StoperPoCisteni.IN.PritomnostPaletky_IS6;

			IF StoperPoCisteni.KoniecCyklu THEN
				SC_StoperPoCisteni.ResetStep:= TRUE;
				SC_StoperPoCisteni.Step:= 0;
			ELSIF SC_StoperPoCisteni.IdleTime.Q THEN
				StoperPoCisteni_Statistika.IN.START_MeraniaCasu:= TRUE;
				StoperPoCisteni_Statistika.IN.ZAPIS_MeraniaCasu:= TRUE;
				SC_StoperPoCisteni.ResetStep:= TRUE;
				SC_StoperPoCisteni.Step:= 101;
			END_IF

		101:
			SC_StoperPoCisteni.StepName:='101 - Automaticky Rezim - cakam na vyvezenie paletky na stoper etiketovania';
			SC_StoperPoCisteni.IdleTime.PT:= T#200ms;
			SC_StoperPoCisteni.AlarmTime.PT:= T#5s;

			IF StoperPoCisteni.KoniecCyklu THEN
				SC_StoperPoCisteni.ResetStep:= TRUE;
				SC_StoperPoCisteni.Step:= 0;
			ELSIF SC_StoperEtiketovania.Step = 100 AND NOT StoperEtiketovania.IN.PritomnostPaletky_IS16 THEN
				SC_StoperPoCisteni.ResetStep:= TRUE;
				SC_StoperPoCisteni.Step:= 105;
			END_IF

		105:
			SC_StoperPoCisteni.StepName:='105 - Automaticky Rezim - vyvazam paletku na stoper etiketovania';
			SC_StoperPoCisteni.IdleTime.PT:= T#4s;
			SC_StoperPoCisteni.AlarmTime.PT:= T#20s;

			IF NOT SC_StoperPoCisteni.Switch1 THEN
				StoperPoCisteni.OUT.StoperZASUN_YV006:= TRUE;
				StoperPoCisteni.STAV.PrebiehaVyvazaniePaletky:= TRUE;
				SC_StoperPoCisteni.AlarmTime.IN:= TRUE;
				SC_StoperPoCisteni.Switch1:= TRUE;
			END_IF

			IF NOT StoperPoCisteni.IN.PritomnostPaletky_IS6 THEN
				StoperPoCisteni.OUT.StoperZASUN_YV006:= FALSE;
				SC_StoperPoCisteni.AlarmTime.IN:= FALSE;
			END_IF

			IF StoperEtiketovania.IN.PritomnostPaletky_IS16 AND NOT StoperPoCisteni.OUT.StoperZASUN_YV006 THEN
				StoperPoCisteni.STAV.PrebiehaVyvazaniePaletky:= FALSE;
				SC_StoperPoCisteni.ResetStep:= TRUE;
				SC_StoperPoCisteni.Step:= 100;
			ELSIF SC_StoperPoCisteni.AlarmTime.Q THEN
				Alarmy[39]:= TRUE;
				PoruchaCistenia:= TRUE;
				SC_StoperPoCisteni.ResetStep:= TRUE;
				SC_StoperPoCisteni.Step:= 0;
			END_IF

			//*******************************************************Manuálny režim*******************************************************************************//
		700:
			SC_StoperPoCisteni.StepName:='700 - Manualny Rezim';
			SC_StoperPoCisteni.IdleTime.PT:= T#8s;
			SC_StoperPoCisteni.AlarmTime.PT:= T#5s;

	END_CASE

END_PROGRAM

PROGRAM _EXIT
	(* Insert code here *)

END_PROGRAM
```

### Program Logical/Program/DopravnikCistenia (IEC)

#### Main.st - Init, cyclic, exit code
```iecst
PROGRAM _INIT
	DopravCistenia.PAR.ZadanaJoggRychlost:= 10;

END_PROGRAM

PROGRAM _CYCLIC

	//Volanie podprogramov//
	OvlMenica;

	//Volanie funkcie SequenceControl//
	SequenceControl(SC:= SC_DopravCistenia);

	//Reset sekcie //
	IF DopravCistenia.Reset THEN
		SC_DopravCistenia.Step:= 0;
		DopravCistenia.Reset:= FALSE;
	ELSIF NOT Safety.STAV.ZonaCS_AKTIVNA THEN
		SC_DopravCistenia.Step:= 0;
	END_IF

	CASE SC_DopravCistenia.Step OF

		0:
			SC_DopravCistenia.StepName:='0 - Nulovanie';
			DopravCistenia.Automat:= FALSE;
			DopravCistenia.KoniecCyklu:= FALSE;
			DopravCistenia.Manual:= FALSE;
			DopravCistenia.STAV.PoINIT:= FALSE;
			SC_OvlMenica.Step:= 0;

			IF Safety.STAV.ZonaCS_AKTIVNA AND Linka.IN.TlakVzduchu_OK_S2 AND NOT NastalaPorucha AND Linka.STAV.Hardware_OK THEN
				SC_DopravCistenia.ResetStep:= TRUE;
				SC_DopravCistenia.Step:= 1;
			END_IF

		1:
			SC_DopravCistenia.StepName:='1 - Cakam na spustenie vyroby';
			DopravCistenia.KoniecCyklu:= FALSE;
			IF DopravCistenia.Automat THEN
				SC_DopravCistenia.Step:= 2;
			ELSIF DopravCistenia.Manual THEN
				SC_DopravCistenia.Step:= 700;
			END_IF

			//********************************************************Inicializácia****************************************************************************//

		2:
			SC_DopravCistenia.StepName:='2 - Inicializacia - cakam na spustenie inicializacie';
			SC_DopravCistenia.IdleTime.PT:= T#500ms;
			SC_DopravCistenia.AlarmTime.PT:= T#5s;

			SC_DopravCistenia.IdleTime.IN:= TRUE;

			IF SC_DopravCistenia.IdleTime.Q THEN
				SC_DopravCistenia.ResetStep:= TRUE;
				SC_DopravCistenia.Step:= 5;
			END_IF

		5:
			SC_DopravCistenia.StepName:='5 - Inicializacia - spustenie dopravnika a ukoncenie inicializacie';
			SC_DopravCistenia.IdleTime.PT:= T#2s;
			SC_DopravCistenia.AlarmTime.PT:= T#5s;

			DopravCistenia.PAR.ZadanaRychlost:= 50;

			IF NOT SC_DopravCistenia.Switch1 AND SC_OvlMenica.Step = 1 THEN
				DopravCistenia.Dopravnik_RUN:= TRUE;
				SC_DopravCistenia.IdleTime.IN:= TRUE;
				SC_DopravCistenia.Switch1:= TRUE;
			END_IF

			IF SC_DopravCistenia.IdleTime.Q THEN
				DopravCistenia.STAV.PoINIT:= TRUE;
				SC_DopravCistenia.ResetStep:= TRUE;
				SC_DopravCistenia.Step:= 100;
			END_IF

			//********************************************************Automatický režim****************************************************************************//

		100:
			SC_DopravCistenia.StepName:='100 - Automaticky Rezim - cakam na vypnutie dopravnika';
			SC_DopravCistenia.IdleTime.PT:= T#200ms;
			SC_DopravCistenia.AlarmTime.PT:= T#5s;

			DopravCistenia.Dopravnik_RUN:= NOT Linka.STAV.Dopravniky_PAUZA;

			IF DopravCistenia.KoniecCyklu AND NOT StoperPredCistenim.Automat AND NOT StoperPoCisteni.Automat AND NOT VstupVytah.Automat THEN
				SC_DopravCistenia.ResetStep:= TRUE;
				SC_DopravCistenia.Step:= 0;
			END_IF

			//*******************************************************Manuálny režim*******************************************************************************//
		700:
			SC_DopravCistenia.StepName:='700 - Manualny Rezim';
			SC_DopravCistenia.IdleTime.PT:= T#8s;
			SC_DopravCistenia.AlarmTime.PT:= T#5s;

	END_CASE

END_PROGRAM

PROGRAM _EXIT
	(* Insert code here *)

END_PROGRAM
```

#### Variables.var - Local variables
```iecst
VAR
	SC_OvlMenica : SequenceControlTyp := (0);
	Chod_VPRED : BOOL := FALSE;
	Chod_VZAD : BOOL := FALSE;
END_VAR
```

#### OvlMenica.st
```iecst
ACTION OvlMenica:

	//CANopen adresa meniča - 32//

	//Volanie funkčného bloku//
	DopravCistenia.MenicDopravnika_FM1();

	//Volanie funkcie SequenceControl//
	SequenceControl(SC:= SC_OvlMenica);

	//Prepnutie meniča do stavu READY//
	IF EDGEPOS(Safety.STAV.SafetyPLC_Nabehlo)THEN
		IF NOT DopravCistenia.MenicDopravnika_FM1.STAV.READY THEN
			DopravCistenia.MenicDopravnika_FM1.CMD.Potvrd_PORUCHU:= TRUE;
		END_IF
	END_IF

	//Parametre meniča//
	DopravCistenia.MenicDopravnika_FM1.PAR.TypKomunikacieProfinet:= 0;
	DopravCistenia.STAV.AktualnaRychlost:= DopravCistenia.MenicDopravnika_FM1.PAR.AktualnaFrekvencia_Hz;
	DopravCistenia.STAV.BUSY:= DopravCistenia.MenicDopravnika_FM1.STAV.RUN;

	CASE SC_OvlMenica.Step OF

		0:
			SC_OvlMenica.StepName:= '0 - Nulovanie';
			Chod_VPRED:= FALSE;
			Chod_VZAD:= FALSE;
			DopravCistenia.Dopravnik_RUN:= FALSE;
			DopravCistenia.MenicDopravnika_FM1.CMD.HOME:= FALSE;
			DopravCistenia.MenicDopravnika_FM1.CMD.Chod_VPRED:= FALSE;
			DopravCistenia.MenicDopravnika_FM1.CMD.Chod_VZAD:= FALSE;

			IF SC_DopravCistenia.Step <> 0 AND DopravCistenia.MenicDopravnika_FM1.STAV.READY AND NOT DopravCistenia.MenicDopravnika_FM1.STAV.PORUCHA THEN
				SC_OvlMenica.ResetStep:= TRUE;
				SC_OvlMenica.Step:= 1;
			END_IF

		1:
			SC_OvlMenica.StepName:= '1 - Rozhodnutie o cinnosti';
			IF Chod_VPRED THEN
				SC_OvlMenica.Step:= 10;
			ELSIF Chod_VZAD THEN
				SC_OvlMenica.Step:= 20;
			ELSIF DopravCistenia.Dopravnik_RUN THEN
				SC_OvlMenica.Step:= 30;
			END_IF

		10:
			SC_OvlMenica.StepName:= '10 - Chod VPRED';
			SC_OvlMenica.IdleTime.PT:= T#3s;
			SC_OvlMenica.AlarmTime.PT:= T#3s;

			IF DopravCistenia.Automat THEN
				DopravCistenia.MenicDopravnika_FM1.PAR.ZadanaFrekvencia_Hz:= DopravCistenia.PAR.ZadanaRychlost;
			ELSE
				DopravCistenia.MenicDopravnika_FM1.PAR.ZadanaFrekvencia_Hz:= DopravCistenia.PAR.ZadanaJoggRychlost;
			END_IF

			IF NOT SC_OvlMenica.Switch1 THEN
				DopravCistenia.MenicDopravnika_FM1.CMD.Chod_VPRED:= TRUE;
				SC_OvlMenica.Switch1:= TRUE;
			END_IF

			IF NOT Chod_VPRED THEN
				SC_OvlMenica.ResetStep:= TRUE;
				SC_OvlMenica.Step:= 0;
			END_IF

		20:
			SC_OvlMenica.StepName:= '20 - Chod VZAD';
			SC_OvlMenica.IdleTime.PT:= T#3s;
			SC_OvlMenica.AlarmTime.PT:= T#3s;

			IF DopravCistenia.Automat THEN
				DopravCistenia.MenicDopravnika_FM1.PAR.ZadanaFrekvencia_Hz:= DopravCistenia.PAR.ZadanaRychlost;
			ELSE
				DopravCistenia.MenicDopravnika_FM1.PAR.ZadanaFrekvencia_Hz:= DopravCistenia.PAR.ZadanaJoggRychlost;
			END_IF

			IF NOT SC_OvlMenica.Switch1 THEN
				DopravCistenia.MenicDopravnika_FM1.CMD.Chod_VZAD:= TRUE;
				SC_OvlMenica.Switch1:= TRUE;
			END_IF

			IF NOT Chod_VZAD THEN
				SC_OvlMenica.ResetStep:= TRUE;
				SC_OvlMenica.Step:= 0;
			END_IF

		30:
			SC_OvlMenica.StepName:= '30 - Chod VPRED v automate';
			SC_OvlMenica.IdleTime.PT:= T#3s;
			SC_OvlMenica.AlarmTime.PT:= T#3s;

			IF DopravCistenia.Automat THEN
				DopravCistenia.MenicDopravnika_FM1.PAR.ZadanaFrekvencia_Hz:= DopravCistenia.PAR.ZadanaRychlost;
			ELSE
				DopravCistenia.MenicDopravnika_FM1.PAR.ZadanaFrekvencia_Hz:= DopravCistenia.PAR.ZadanaJoggRychlost;
			END_IF

			IF NOT SC_OvlMenica.Switch1 THEN
				DopravCistenia.MenicDopravnika_FM1.CMD.Chod_VPRED:= TRUE;
				SC_OvlMenica.Switch1:= TRUE;
			END_IF

			IF NOT DopravCistenia.Dopravnik_RUN THEN
				SC_OvlMenica.ResetStep:= TRUE;
				SC_OvlMenica.Step:= 0;
			END_IF

	END_CASE

END_ACTION
```

### Program Logical/Program/StoperEtiketovania (IEC)
